   cmFinalRollerRearAxisX.commandConfiguration.phasing.phaseShiftChangeOnTheFly := FALSE;
   cmFinalRollerRearAxisX.commandConfiguration.offset.offset := 0.0;
   cmFinalRollerRearAxisX.commandConfiguration.offset.profileReference := 1;
   cmFinalRollerRearAxisX.commandConfiguration.offset.offsetDistance := 0.0;
   cmFinalRollerRearAxisX.commandConfiguration.offset.startPosition := 0.0;
   cmFinalRollerRearAxisX.commandConfiguration.offset.direction := 3;
   cmFinalRollerRearAxisX.commandConfiguration.offset.offsetAbsolute := TRUE;
   cmFinalRollerRearAxisX.commandConfiguration.offset.offsetChangeOnTheFly := FALSE;
   cmFinalRollerRearAxisX.commands.enableMasterControl := TRUE;
   cmFinalRollerRearAxisX.commands.enableAxis := FALSE;
   cmFinalRollerRearAxisX.commands.resetAxis := FALSE;
   cmFinalRollerRearAxisX.commands.openBrake := FALSE;
   cmFinalRollerRearAxisX.commands.jogForward := FALSE;
   cmFinalRollerRearAxisX.commands.jogBackward := FALSE;
   cmFinalRollerRearAxisX.commands.moveVelocity := FALSE;
   cmFinalRollerRearAxisX.commands.stop := FALSE;
   cmFinalRollerRearAxisX.commands.fastStop := FALSE;
   cmFinalRollerRearAxisX.commands.torqueLimiting := FALSE;
   cmFinalRollerRearAxisX.commands.homing := FALSE;
   cmFinalRollerRearAxisX.commands.posRelative := FALSE;
   cmFinalRollerRearAxisX.commands.posAbsolute := FALSE;
   cmFinalRollerRearAxisX.commands.posSuperimposed := FALSE;
   cmFinalRollerRearAxisX.commands.haltSuperimposed := FALSE;
   cmFinalRollerRearAxisX.commands.selectSetPosition := 0;
   cmFinalRollerRearAxisX.commands.uploadParameters := FALSE;
   cmFinalRollerRearAxisX.commands.refreshConfiguration := FALSE;
   cmFinalRollerRearAxisX.commands.editConfiguration := FALSE;
   cmFinalRollerRearAxisX.commands.saveConfiguration := FALSE;
   cmFinalRollerRearAxisX.commands.uploadCurrentTorque := FALSE;
   cmFinalRollerRearAxisX.commands.reset := FALSE;
   cmFinalRollerRearAxisX.monitoring.enable := TRUE;
   cmFinalRollerRearAxisX.monitoring.referenceDesignator := WSTRING#'FinalRollerRearAxisX';
   cmFinalRollerRearAxisX.monitoring.enabled := TRUE;
   cmFinalRollerRearAxisX.monitoring.enableManualCmds := FALSE;
   cmFinalRollerRearAxisX.monitoring.reset := FALSE;
   cmFinalRollerRearAxisX.monitoring.resetAxis := FALSE;
   cmFinalRollerRearAxisX.monitoring.enableAxis := TRUE;
   cmFinalRollerRearAxisX.monitoring.openBrake := FALSE;
   cmFinalRollerRearAxisX.monitoring.jogBackward := FALSE;
   cmFinalRollerRearAxisX.monitoring.jogForward := FALSE;
   cmFinalRollerRearAxisX.monitoring.moveVelocity := FALSE;
   cmFinalRollerRearAxisX.monitoring.stop := FALSE;
   cmFinalRollerRearAxisX.monitoring.fastStop := FALSE;
   cmFinalRollerRearAxisX.monitoring.torqueLimiting := FALSE;
   cmFinalRollerRearAxisX.monitoring.homing := FALSE;
   cmFinalRollerRearAxisX.monitoring.posRelative := FALSE;
   cmFinalRollerRearAxisX.monitoring.posAbsolute := FALSE;
   cmFinalRollerRearAxisX.monitoring.posSuperimposed := FALSE;
   cmFinalRollerRearAxisX.monitoring.haltSuperimposed := FALSE;
   cmFinalRollerRearAxisX.monitoring.brakeOpened := FALSE;
   cmFinalRollerRearAxisX.monitoring.axisEnabled := TRUE;
   cmFinalRollerRearAxisX.monitoring.resetActive := FALSE;
   cmFinalRollerRearAxisX.monitoring.inVelocity := FALSE;
   cmFinalRollerRearAxisX.monitoring.inLimitation := FALSE;
   cmFinalRollerRearAxisX.monitoring.inClamping := FALSE;
   cmFinalRollerRearAxisX.monitoring.startSync := FALSE;
   cmFinalRollerRearAxisX.monitoring.inSync := FALSE;
   cmFinalRollerRearAxisX.monitoring.inSimulation := FALSE;
   cmFinalRollerRearAxisX.monitoring.jogSelected := FALSE;
   cmFinalRollerRearAxisX.monitoring.moveVelocitySelected := FALSE;
   cmFinalRollerRearAxisX.monitoring.stopSelected := FALSE;
   cmFinalRollerRearAxisX.monitoring.fastStopSelected := FALSE;
   cmFinalRollerRearAxisX.monitoring.torqueLimitingSelected := FALSE;
   cmFinalRollerRearAxisX.monitoring.homingSelected := FALSE;
   cmFinalRollerRearAxisX.monitoring.posRelativeSelected := FALSE;
   cmFinalRollerRearAxisX.monitoring.posAbsoluteSelected := FALSE;
   cmFinalRollerRearAxisX.monitoring.posSuperimposedSelected := FALSE;
   cmFinalRollerRearAxisX.monitoring.haltSuperimposedSelected := FALSE;
   cmFinalRollerRearAxisX.monitoring.commandBusy := FALSE;
   cmFinalRollerRearAxisX.monitoring.commandDone := FALSE;
   cmFinalRollerRearAxisX.monitoring.commandAborted := FALSE;
   cmFinalRollerRearAxisX.monitoring.homingCommandBusy := FALSE;
   cmFinalRollerRearAxisX.monitoring.homingCommandDone := FALSE;
   cmFinalRollerRearAxisX.monitoring.homingCommandAborted := FALSE;
   cmFinalRollerRearAxisX.monitoring.superimposedBusy := FALSE;
   cmFinalRollerRearAxisX.monitoring.superimposedDone := FALSE;
   cmFinalRollerRearAxisX.monitoring.superimposedAborted := FALSE;
   cmFinalRollerRearAxisX.monitoring.selectSetPosition := 0;
   cmFinalRollerRearAxisX.monitoring.selectionController := FALSE;
   cmFinalRollerRearAxisX.monitoring.interlockGeneral := TRUE;
   cmFinalRollerRearAxisX.monitoring.interlockJogForward := TRUE;
   cmFinalRollerRearAxisX.monitoring.interlockJogBackward := TRUE;
   cmFinalRollerRearAxisX.monitoring.interlockWarningGeneral := FALSE;
   cmFinalRollerRearAxisX.monitoring.interlockWarningJogForward := FALSE;
   cmFinalRollerRearAxisX.monitoring.interlockWarningJogBackward := FALSE;
   cmFinalRollerRearAxisX.monitoring.valid := TRUE;
   cmFinalRollerRearAxisX.monitoring.busy := TRUE;
   cmFinalRollerRearAxisX.monitoring.error := FALSE;
   cmFinalRollerRearAxisX.monitoring.status := 16#7002;
   cmFinalRollerRearAxisX.monitoring.subfunctionStatus := 16#0000;
   cmFinalRollerRearAxisX.monitoring.actualPosition := 0.0;
   cmFinalRollerRearAxisX.monitoring.actualSpeed := 0.0;
   cmFinalRollerRearAxisX.monitoring.speedUnit := 1062;
   cmFinalRollerRearAxisX.monitoring.positionUnit := 1013;
   cmFinalRollerRearAxisX.monitoring.axisStatus1 := 16#0200_10E1;
   cmFinalRollerRearAxisX.monitoring.axisStatus2 := 16#0000_0000;
   cmFinalRollerRearAxisX.monitoring.axisType := 1;
   cmFinalRollerRearAxisX.monitoring.maxVelocity := 2500.0;
   cmFinalRollerRearAxisX.monitoring.actualCurrent := 0.0;
   cmFinalRollerRearAxisX.monitoring.actualTorque := 0.0;
   cmFinalRollerRearAxisX.monitoring.velocityOverrideEnabled := FALSE;
   cmFinalRollerRearAxisX.monitoring.sinaParaError := FALSE;
   cmFinalRollerRearAxisX.monitoring.sinaParaStatus := 16#0000_0000;
   cmFinalRollerRearAxisX.configuration.referenceDesignator := WSTRING#'FinalRollerRearAxisX';
   cmFinalRollerRearAxisX.configuration.disableAlarms := FALSE;
   cmFinalRollerRearAxisX.configuration.masterControlPopUp := TRUE;
   cmFinalRollerRearAxisX.configuration.setPositions[0].position := 0.0;
   cmFinalRollerRearAxisX.configuration.setPositions[1].position := 500.0;
   cmFinalRollerRearAxisX.configuration.setPositions[2..15].position := 0.0;
   cmFinalRollerRearAxisX.configuration.setPositions[0..1].velocity := 500.0;
   cmFinalRollerRearAxisX.configuration.setPositions[2..15].velocity := -1.0;
   cmFinalRollerRearAxisX.configuration.setPositions[0..1].acceleration := 5000.0;
   cmFinalRollerRearAxisX.configuration.setPositions[2..15].acceleration := -1.0;
   cmFinalRollerRearAxisX.configuration.setPositions[0..1].deceleration := 5000.0;
   cmFinalRollerRearAxisX.configuration.setPositions[2..15].deceleration := -1.0;
   cmFinalRollerRearAxisX.configuration.setPositions[0..15]."name" := '';
   cmMendrelAnodeFrontAxisY.commandConfiguration.generalSettings.stopOnError := TRUE;
   cmMendrelAnodeFrontAxisY.commandConfiguration.generalSettings.resetWithRestart := FALSE;
   cmMendrelAnodeFrontAxisY.commandConfiguration.generalSettings.abortWaitingSyncCmd := TRUE;
   cmMendrelAnodeFrontAxisY.commandConfiguration.power.startMode := 1;
   cmMendrelAnodeFrontAxisY.commandConfiguration.power.stopMode := 0;
   cmMendrelAnodeFrontAxisY.commandConfiguration.power.syncMotionSimulation := FALSE;
   cmMendrelAnodeFrontAxisY.commandConfiguration.power.syncMotionSimulationExtendedMode := -1;
   cmMendrelAnodeFrontAxisY.commandConfiguration.jog.velocity := 0.0;
   cmMendrelAnodeFrontAxisY.commandConfiguration.jog.acceleration := -1.0;
   cmMendrelAnodeFrontAxisY.commandConfiguration.jog.deceleration := -1.0;
   cmMendrelAnodeFrontAxisY.commandConfiguration.jog.jerk := -1.0;
   cmMendrelAnodeFrontAxisY.commandConfiguration.jog.positionControlled := TRUE;
   cmMendrelAnodeFrontAxisY.commandConfiguration.jog.increment := 0.0;
   cmMendrelAnodeFrontAxisY.commandConfiguration.jog.mode := 0;
   cmMendrelAnodeFrontAxisY.commandConfiguration.moveVelocity.velocity := 0.0;
   cmMendrelAnodeFrontAxisY.commandConfiguration.moveVelocity.acceleration := -1.0;
   cmMendrelAnodeFrontAxisY.commandConfiguration.moveVelocity.deceleration := -1.0;
   cmMendrelAnodeFrontAxisY.commandConfiguration.moveVelocity.jerk := -1.0;
   cmMendrelAnodeFrontAxisY.commandConfiguration.moveVelocity.direction := 0;
   cmMendrelAnodeFrontAxisY.commandConfiguration.moveVelocity.positionControlled := TRUE;
   cmMendrelAnodeFrontAxisY.commandConfiguration.moveVelocity.velocityChangeOnTheFly := FALSE;
   cmMendrelAnodeFrontAxisY.commandConfiguration.stop.deceleration := -1.0;
   cmMendrelAnodeFrontAxisY.commandConfiguration.stop.jerk := -1.0;
   cmMendrelAnodeFrontAxisY.commandConfiguration.stop.abortAcceleration := FALSE;
   cmMendrelAnodeFrontAxisY.commandConfiguration.fastStop.deceleration := -1.0;
   cmMendrelAnodeFrontAxisY.commandConfiguration.fastStop.jerk := -1.0;
   cmMendrelAnodeFrontAxisY.commandConfiguration.fastStop.abortAcceleration := FALSE;
   cmMendrelAnodeFrontAxisY.commandConfiguration.fastStop.replaceStopPossible := FALSE;
   cmMendrelAnodeFrontAxisY.commandConfiguration.torqueLimiting.limit := -1.0;
   cmMendrelAnodeFrontAxisY.commandConfiguration.torqueLimiting.mode := 0;
   cmMendrelAnodeFrontAxisY.commandConfiguration.homing.position := 0.0;
   cmMendrelAnodeFrontAxisY.commandConfiguration.homing.mode := 0;
   cmMendrelAnodeFrontAxisY.commandConfiguration.homing.sensor := 0;
   cmMendrelAnodeFrontAxisY.commandConfiguration.homing.extendedMode := -1;
   cmMendrelAnodeFrontAxisY.commandConfiguration.homing.extendedModeTorqueLimit := 0.0;
   cmMendrelAnodeFrontAxisY.commandConfiguration.homing.extendedModeTargetPosition := 0.0;
   cmMendrelAnodeFrontAxisY.commandConfiguration.posRelative.distance := 0.0;
   cmMendrelAnodeFrontAxisY.commandConfiguration.posRelative.velocity := -1.0;
   cmMendrelAnodeFrontAxisY.commandConfiguration.posRelative.acceleration := -1.0;
   cmMendrelAnodeFrontAxisY.commandConfiguration.posRelative.deceleration := -1.0;
   cmMendrelAnodeFrontAxisY.commandConfiguration.posRelative.jerk := -1.0;
   cmMendrelAnodeFrontAxisY.commandConfiguration.posRelative.direction := 0;
   cmMendrelAnodeFrontAxisY.commandConfiguration.posAbsolute.position := 0.0;
   cmMendrelAnodeFrontAxisY.commandConfiguration.posAbsolute.velocity := -1.0;
   cmMendrelAnodeFrontAxisY.commandConfiguration.posAbsolute.acceleration := -1.0;
   cmMendrelAnodeFrontAxisY.commandConfiguration.posAbsolute.deceleration := -1.0;
   cmMendrelAnodeFrontAxisY.commandConfiguration.posAbsolute.jerk := -1.0;
   cmMendrelAnodeFrontAxisY.commandConfiguration.posAbsolute.direction := 1;
   cmMendrelAnodeFrontAxisY.commandConfiguration.posAbsolute.positionChangeOnTheFly := FALSE;
   cmMendrelAnodeFrontAxisY.commandConfiguration.posAbsolute.velocityChangeOnTheFly := FALSE;
   cmMendrelAnodeFrontAxisY.commandConfiguration.posSuperimposed.distance := 0.0;
   cmMendrelAnodeFrontAxisY.commandConfiguration.posSuperimposed.velocityDiff := -1.0;
   cmMendrelAnodeFrontAxisY.commandConfiguration.posSuperimposed.acceleration := -1.0;
   cmMendrelAnodeFrontAxisY.commandConfiguration.posSuperimposed.deceleration := -1.0;
   cmMendrelAnodeFrontAxisY.commandConfiguration.posSuperimposed.jerk := -1.0;
   cmMendrelAnodeFrontAxisY.commandConfiguration.posSuperimposed.direction := 0;
   cmMendrelAnodeFrontAxisY.commandConfiguration.haltSuperimposed.deceleration := -1.0;
   cmMendrelAnodeFrontAxisY.commandConfiguration.haltSuperimposed.jerk := -1.0;
   cmMendrelAnodeFrontAxisY.commandConfiguration.haltSuperimposed.abortAcceleration := FALSE;
   cmMendrelAnodeFrontAxisY.commandConfiguration.gearInRelative.ratioNumerator := 1;
   cmMendrelAnodeFrontAxisY.commandConfiguration.gearInRelative.ratioDenominator := 1;
   cmMendrelAnodeFrontAxisY.commandConfiguration.gearInRelative.acceleration := -1.0;
   cmMendrelAnodeFrontAxisY.commandConfiguration.gearInRelative.deceleration := -1.0;
   cmMendrelAnodeFrontAxisY.commandConfiguration.gearInRelative.jerk := -1.0;
   cmMendrelAnodeFrontAxisY.commandConfiguration.gearInRelative.ratioChangeOnTheFly := FALSE;
   cmMendrelAnodeFrontAxisY.commandConfiguration.gearInAbsolute.ratioNumerator := 1;
   cmMendrelAnodeFrontAxisY.commandConfiguration.gearInAbsolute.ratioDenominator := 1;
   cmMendrelAnodeFrontAxisY.commandConfiguration.gearInAbsolute.masterSyncPosition := 0.0;
   cmMendrelAnodeFrontAxisY.commandConfiguration.gearInAbsolute.slaveSyncPosition := 0.0;
   cmMendrelAnodeFrontAxisY.commandConfiguration.gearInAbsolute.syncProfileReference := 1;
   cmMendrelAnodeFrontAxisY.commandConfiguration.gearInAbsolute.masterStartDistance := 0.0;
   cmMendrelAnodeFrontAxisY.commandConfiguration.gearInAbsolute.velocity := -1.0;
   cmMendrelAnodeFrontAxisY.commandConfiguration.gearInAbsolute.acceleration := -1.0;
   cmMendrelAnodeFrontAxisY.commandConfiguration.gearInAbsolute.deceleration := -1.0;
   cmMendrelAnodeFrontAxisY.commandConfiguration.gearInAbsolute.jerk := -1.0;
   cmMendrelAnodeFrontAxisY.commandConfiguration.gearInAbsolute.syncDirection := 1;
   cmMendrelAnodeFrontAxisY.commandConfiguration.gearInAbsolute.ratioChangeOnTheFly := FALSE;
   cmMendrelAnodeFrontAxisY.commandConfiguration.gearInVelocity.continuousUpdate := FALSE;
   cmMendrelAnodeFrontAxisY.commandConfiguration.gearInVelocity.ratioNumerator := 1;
   cmMendrelAnodeFrontAxisY.commandConfiguration.gearInVelocity.ratioDenominator := 1;
   cmMendrelAnodeFrontAxisY.commandConfiguration.gearInVelocity.acceleration := -1.0;
   cmMendrelAnodeFrontAxisY.commandConfiguration.gearInVelocity.deceleration := -1.0;
   cmMendrelAnodeFrontAxisY.commandConfiguration.gearInVelocity.jerk := -1.0;
   cmMendrelAnodeFrontAxisY.commandConfiguration.gearInVelocity.positionControlled := FALSE;
   cmMendrelAnodeFrontAxisY.commandConfiguration.camIn.masterOffset := 0.0;
   cmMendrelAnodeFrontAxisY.commandConfiguration.camIn.slaveOffset := 0.0;
   cmMendrelAnodeFrontAxisY.commandConfiguration.camIn.masterScaling := 1.0;
   cmMendrelAnodeFrontAxisY.commandConfiguration.camIn.slaveScaling := 1.0;
   cmMendrelAnodeFrontAxisY.commandConfiguration.camIn.masterSyncPosition := 0.0;
   cmMendrelAnodeFrontAxisY.commandConfiguration.camIn.syncProfileReference := 1;
   cmMendrelAnodeFrontAxisY.commandConfiguration.camIn.masterStartDistance := 0.0;
   cmMendrelAnodeFrontAxisY.commandConfiguration.camIn.velocity := -1.0;
   cmMendrelAnodeFrontAxisY.commandConfiguration.camIn.acceleration := -1.0;
   cmMendrelAnodeFrontAxisY.commandConfiguration.camIn.deceleration := -1.0;
   cmMendrelAnodeFrontAxisY.commandConfiguration.camIn.jerk := -1.0;
   cmMendrelAnodeFrontAxisY.commandConfiguration.camIn.applicationMode := 0;
   cmMendrelAnodeFrontAxisY.commandConfiguration.camIn.syncDirection := 1;
   cmMendrelAnodeFrontAxisY.commandConfiguration.gearOutCamOut.slavePosition := 0.0;
   cmMendrelAnodeFrontAxisY.commandConfiguration.gearOutCamOut.syncProfileReference := 1;
   cmMendrelAnodeFrontAxisY.commandConfiguration.gearOutCamOut.masterStopDistance := 0.0;
   cmMendrelAnodeFrontAxisY.commandConfiguration.gearOutCamOut.deceleration := -1.0;
   cmMendrelAnodeFrontAxisY.commandConfiguration.gearOutCamOut.jerk := -1.0;
   cmMendrelAnodeFrontAxisY.commandConfiguration.gearOutCamOut.syncOutDirection := 3;
   cmMendrelAnodeFrontAxisY.commandConfiguration.gearOutCamOut.gearOutCamOutMode := -1;
   cmMendrelAnodeFrontAxisY.commandConfiguration.phasing.phaseShift := 0.0;
   cmMendrelAnodeFrontAxisY.commandConfiguration.phasing.velocity := -1.0;
   cmMendrelAnodeFrontAxisY.commandConfiguration.phasing.acceleration := -1.0;
   cmMendrelAnodeFrontAxisY.commandConfiguration.phasing.deceleration := -1.0;
   cmMendrelAnodeFrontAxisY.commandConfiguration.phasing.jerk := -1.0;
   cmMendrelAnodeFrontAxisY.commandConfiguration.phasing.profileReference := 0;
   cmMendrelAnodeFrontAxisY.commandConfiguration.phasing.phasingDistance := 0.0;
   cmMendrelAnodeFrontAxisY.commandConfiguration.phasing.startPosition := 0.0;
   cmMendrelAnodeFrontAxisY.commandConfiguration.phasing.direction := 3;
   cmMendrelAnodeFrontAxisY.commandConfiguration.phasing.phaseAbsolute := TRUE;
   cmMendrelAnodeFrontAxisY.commandConfiguration.phasing.phaseShiftChangeOnTheFly := FALSE;
   cmMendrelAnodeFrontAxisY.commandConfiguration.offset.offset := 0.0;
   cmMendrelAnodeFrontAxisY.commandConfiguration.offset.profileReference := 1;
   cmMendrelAnodeFrontAxisY.commandConfiguration.offset.offsetDistance := 0.0;
   cmMendrelAnodeFrontAxisY.commandConfiguration.offset.startPosition := 0.0;
   cmMendrelAnodeFrontAxisY.commandConfiguration.offset.direction := 3;
   cmMendrelAnodeFrontAxisY.commandConfiguration.offset.offsetAbsolute := TRUE;
   cmMendrelAnodeFrontAxisY.commandConfiguration.offset.offsetChangeOnTheFly := FALSE;
   cmMendrelAnodeFrontAxisY.commands.enableMasterControl := TRUE;
   cmMendrelAnodeFrontAxisY.commands.enableAxis := FALSE;
   cmMendrelAnodeFrontAxisY.commands.resetAxis := FALSE;
   cmMendrelAnodeFrontAxisY.commands.openBrake := FALSE;
   cmMendrelAnodeFrontAxisY.commands.jogForward := FALSE;
   cmMendrelAnodeFrontAxisY.commands.jogBackward := FALSE;
   cmMendrelAnodeFrontAxisY.commands.moveVelocity := FALSE;
   cmMendrelAnodeFrontAxisY.commands.stop := FALSE;
   cmMendrelAnodeFrontAxisY.commands.fastStop := FALSE;
   cmMendrelAnodeFrontAxisY.commands.torqueLimiting := FALSE;
   cmMendrelAnodeFrontAxisY.commands.homing := FALSE;
   cmMendrelAnodeFrontAxisY.commands.posRelative := FALSE;
   cmMendrelAnodeFrontAxisY.commands.posAbsolute := FALSE;
   cmMendrelAnodeFrontAxisY.commands.posSuperimposed := FALSE;
   cmMendrelAnodeFrontAxisY.commands.haltSuperimposed := FALSE;
   cmMendrelAnodeFrontAxisY.commands.selectSetPosition := 1;
   cmMendrelAnodeFrontAxisY.commands.uploadParameters := FALSE;
   cmMendrelAnodeFrontAxisY.commands.refreshConfiguration := FALSE;
   cmMendrelAnodeFrontAxisY.commands.editConfiguration := FALSE;
   cmMendrelAnodeFrontAxisY.commands.saveConfiguration := FALSE;
   cmMendrelAnodeFrontAxisY.commands.uploadCurrentTorque := FALSE;
   cmMendrelAnodeFrontAxisY.commands.reset := FALSE;
   cmMendrelAnodeFrontAxisY.monitoring.enable := TRUE;
   cmMendrelAnodeFrontAxisY.monitoring.referenceDesignator := WSTRING#'MendrelAnodeFrontAxisY';
   cmMendrelAnodeFrontAxisY.monitoring.enabled := TRUE;
   cmMendrelAnodeFrontAxisY.monitoring.enableManualCmds := FALSE;
   cmMendrelAnodeFrontAxisY.monitoring.reset := FALSE;
   cmMendrelAnodeFrontAxisY.monitoring.resetAxis := FALSE;
   cmMendrelAnodeFrontAxisY.monitoring.enableAxis := TRUE;
   cmMendrelAnodeFrontAxisY.monitoring.openBrake := FALSE;
   cmMendrelAnodeFrontAxisY.monitoring.jogBackward := FALSE;
   cmMendrelAnodeFrontAxisY.monitoring.jogForward := FALSE;
   cmMendrelAnodeFrontAxisY.monitoring.moveVelocity := FALSE;
   cmMendrelAnodeFrontAxisY.monitoring.stop := FALSE;
   cmMendrelAnodeFrontAxisY.monitoring.fastStop := FALSE;
   cmMendrelAnodeFrontAxisY.monitoring.torqueLimiting := FALSE;
   cmMendrelAnodeFrontAxisY.monitoring.homing := FALSE;
   cmMendrelAnodeFrontAxisY.monitoring.posRelative := FALSE;
   cmMendrelAnodeFrontAxisY.monitoring.posAbsolute := FALSE;
   cmMendrelAnodeFrontAxisY.monitoring.posSuperimposed := FALSE;
   cmMendrelAnodeFrontAxisY.monitoring.haltSuperimposed := FALSE;
   cmMendrelAnodeFrontAxisY.monitoring.brakeOpened := FALSE;
   cmMendrelAnodeFrontAxisY.monitoring.axisEnabled := TRUE;
   cmMendrelAnodeFrontAxisY.monitoring.resetActive := FALSE;
   cmMendrelAnodeFrontAxisY.monitoring.inVelocity := FALSE;
   cmMendrelAnodeFrontAxisY.monitoring.inLimitation := FALSE;
   cmMendrelAnodeFrontAxisY.monitoring.inClamping := FALSE;
   cmMendrelAnodeFrontAxisY.monitoring.startSync := FALSE;
   cmMendrelAnodeFrontAxisY.monitoring.inSync := FALSE;
   cmMendrelAnodeFrontAxisY.monitoring.inSimulation := FALSE;
   cmMendrelAnodeFrontAxisY.monitoring.jogSelected := FALSE;
   cmMendrelAnodeFrontAxisY.monitoring.moveVelocitySelected := FALSE;
   cmMendrelAnodeFrontAxisY.monitoring.stopSelected := FALSE;
   cmMendrelAnodeFrontAxisY.monitoring.fastStopSelected := FALSE;
   cmMendrelAnodeFrontAxisY.monitoring.torqueLimitingSelected := FALSE;
   cmMendrelAnodeFrontAxisY.monitoring.homingSelected := FALSE;
   cmMendrelAnodeFrontAxisY.monitoring.posRelativeSelected := FALSE;
   cmMendrelAnodeFrontAxisY.monitoring.posAbsoluteSelected := FALSE;
   cmMendrelAnodeFrontAxisY.monitoring.posSuperimposedSelected := FALSE;
   cmMendrelAnodeFrontAxisY.monitoring.haltSuperimposedSelected := FALSE;
   cmMendrelAnodeFrontAxisY.monitoring.commandBusy := FALSE;
   cmMendrelAnodeFrontAxisY.monitoring.commandDone := FALSE;
   cmMendrelAnodeFrontAxisY.monitoring.commandAborted := FALSE;
   cmMendrelAnodeFrontAxisY.monitoring.homingCommandBusy := FALSE;
   cmMendrelAnodeFrontAxisY.monitoring.homingCommandDone := FALSE;
   cmMendrelAnodeFrontAxisY.monitoring.homingCommandAborted := FALSE;
   cmMendrelAnodeFrontAxisY.monitoring.superimposedBusy := FALSE;
   cmMendrelAnodeFrontAxisY.monitoring.superimposedDone := FALSE;
   cmMendrelAnodeFrontAxisY.monitoring.superimposedAborted := FALSE;
   cmMendrelAnodeFrontAxisY.monitoring.selectSetPosition := 1;
   cmMendrelAnodeFrontAxisY.monitoring.selectionController := FALSE;
   cmMendrelAnodeFrontAxisY.monitoring.interlockGeneral := TRUE;
   cmMendrelAnodeFrontAxisY.monitoring.interlockJogForward := TRUE;
   cmMendrelAnodeFrontAxisY.monitoring.interlockJogBackward := TRUE;
   cmMendrelAnodeFrontAxisY.monitoring.interlockWarningGeneral := FALSE;
   cmMendrelAnodeFrontAxisY.monitoring.interlockWarningJogForward := FALSE;
   cmMendrelAnodeFrontAxisY.monitoring.interlockWarningJogBackward := FALSE;
   cmMendrelAnodeFrontAxisY.monitoring.valid := TRUE;
   cmMendrelAnodeFrontAxisY.monitoring.busy := TRUE;
   cmMendrelAnodeFrontAxisY.monitoring.error := FALSE;
   cmMendrelAnodeFrontAxisY.monitoring.status := 16#7002;
   cmMendrelAnodeFrontAxisY.monitoring.subfunctionStatus := 16#0000;
   cmMendrelAnodeFrontAxisY.monitoring.actualPosition := 50.0;
   cmMendrelAnodeFrontAxisY.monitoring.actualSpeed := 0.0;
   cmMendrelAnodeFrontAxisY.monitoring.speedUnit := 1062;
   cmMendrelAnodeFrontAxisY.monitoring.positionUnit := 1013;
   cmMendrelAnodeFrontAxisY.monitoring.axisStatus1 := 16#0240_10A1;
   cmMendrelAnodeFrontAxisY.monitoring.axisStatus2 := 16#0000_0000;
   cmMendrelAnodeFrontAxisY.monitoring.axisType := 1;
   cmMendrelAnodeFrontAxisY.monitoring.maxVelocity := 2500.0;
   cmMendrelAnodeFrontAxisY.monitoring.actualCurrent := 0.0;
   cmMendrelAnodeFrontAxisY.monitoring.actualTorque := 0.0;
   cmMendrelAnodeFrontAxisY.monitoring.velocityOverrideEnabled := FALSE;
   cmMendrelAnodeFrontAxisY.monitoring.sinaParaError := FALSE;
   cmMendrelAnodeFrontAxisY.monitoring.sinaParaStatus := 16#0000_0000;
   cmMendrelAnodeFrontAxisY.configuration.referenceDesignator := WSTRING#'MendrelAnodeFrontAxisY';
   cmMendrelAnodeFrontAxisY.configuration.disableAlarms := FALSE;
   cmMendrelAnodeFrontAxisY.configuration.masterControlPopUp := TRUE;
   cmMendrelAnodeFrontAxisY.configuration.setPositions[0].position := 0.0;
   cmMendrelAnodeFrontAxisY.configuration.setPositions[1].position := 50.0;
   cmMendrelAnodeFrontAxisY.configuration.setPositions[2..15].position := 0.0;
   cmMendrelAnodeFrontAxisY.configuration.setPositions[0..1].velocity := 50.0;
   cmMendrelAnodeFrontAxisY.configuration.setPositions[2..15].velocity := -1.0;
   cmMendrelAnodeFrontAxisY.configuration.setPositions[0..1].acceleration := 500.0;
   cmMendrelAnodeFrontAxisY.configuration.setPositions[2..15].acceleration := -1.0;
   cmMendrelAnodeFrontAxisY.configuration.setPositions[0..1].deceleration := 500.0;
   cmMendrelAnodeFrontAxisY.configuration.setPositions[2..15].deceleration := -1.0;
   cmMendrelAnodeFrontAxisY.configuration.setPositions[0..15]."name" := '';
   cmMendrelAnodeFrontAxisZ.commandConfiguration.generalSettings.stopOnError := TRUE;
   cmMendrelAnodeFrontAxisZ.commandConfiguration.generalSettings.resetWithRestart := FALSE;
   cmMendrelAnodeFrontAxisZ.commandConfiguration.generalSettings.abortWaitingSyncCmd := TRUE;
   cmMendrelAnodeFrontAxisZ.commandConfiguration.power.startMode := 1;
   cmMendrelAnodeFrontAxisZ.commandConfiguration.power.stopMode := 0;
   cmMendrelAnodeFrontAxisZ.commandConfiguration.power.syncMotionSimulation := FALSE;
   cmMendrelAnodeFrontAxisZ.commandConfiguration.power.syncMotionSimulationExtendedMode := -1;
   cmMendrelAnodeFrontAxisZ.commandConfiguration.jog.velocity := 0.0;
   cmMendrelAnodeFrontAxisZ.commandConfiguration.jog.acceleration := -1.0;
   cmMendrelAnodeFrontAxisZ.commandConfiguration.jog.deceleration := -1.0;
   cmMendrelAnodeFrontAxisZ.commandConfiguration.jog.jerk := -1.0;
   cmMendrelAnodeFrontAxisZ.commandConfiguration.jog.positionControlled := TRUE;
   cmMendrelAnodeFrontAxisZ.commandConfiguration.jog.increment := 0.0;
   cmMendrelAnodeFrontAxisZ.commandConfiguration.jog.mode := 0;
   cmMendrelAnodeFrontAxisZ.commandConfiguration.moveVelocity.velocity := 0.0;
   cmMendrelAnodeFrontAxisZ.commandConfiguration.moveVelocity.acceleration := -1.0;
   cmMendrelAnodeFrontAxisZ.commandConfiguration.moveVelocity.deceleration := -1.0;
   cmMendrelAnodeFrontAxisZ.commandConfiguration.moveVelocity.jerk := -1.0;
   cmMendrelAnodeFrontAxisZ.commandConfiguration.moveVelocity.direction := 0;
   cmMendrelAnodeFrontAxisZ.commandConfiguration.moveVelocity.positionControlled := TRUE;
   cmMendrelAnodeFrontAxisZ.commandConfiguration.moveVelocity.velocityChangeOnTheFly := FALSE;
   cmMendrelAnodeFrontAxisZ.commandConfiguration.stop.deceleration := -1.0;
   cmMendrelAnodeFrontAxisZ.commandConfiguration.stop.jerk := -1.0;
   cmMendrelAnodeFrontAxisZ.commandConfiguration.stop.abortAcceleration := FALSE;
   cmMendrelAnodeFrontAxisZ.commandConfiguration.fastStop.deceleration := -1.0;
   cmMendrelAnodeFrontAxisZ.commandConfiguration.fastStop.jerk := -1.0;
   cmMendrelAnodeFrontAxisZ.commandConfiguration.fastStop.abortAcceleration := FALSE;
   cmMendrelAnodeFrontAxisZ.commandConfiguration.fastStop.replaceStopPossible := FALSE;
   cmMendrelAnodeFrontAxisZ.commandConfiguration.torqueLimiting.limit := -1.0;
   cmMendrelAnodeFrontAxisZ.commandConfiguration.torqueLimiting.mode := 0;
   cmMendrelAnodeFrontAxisZ.commandConfiguration.homing.position := 0.0;
   cmMendrelAnodeFrontAxisZ.commandConfiguration.homing.mode := 0;
   cmMendrelAnodeFrontAxisZ.commandConfiguration.homing.sensor := 0;
   cmMendrelAnodeFrontAxisZ.commandConfiguration.homing.extendedMode := -1;
   cmMendrelAnodeFrontAxisZ.commandConfiguration.homing.extendedModeTorqueLimit := 0.0;
   cmMendrelAnodeFrontAxisZ.commandConfiguration.homing.extendedModeTargetPosition := 0.0;
   cmMendrelAnodeFrontAxisZ.commandConfiguration.posRelative.distance := 0.0;
   cmMendrelAnodeFrontAxisZ.commandConfiguration.posRelative.velocity := -1.0;
   cmMendrelAnodeFrontAxisZ.commandConfiguration.posRelative.acceleration := -1.0;
   cmMendrelAnodeFrontAxisZ.commandConfiguration.posRelative.deceleration := -1.0;
   cmMendrelAnodeFrontAxisZ.commandConfiguration.posRelative.jerk := -1.0;
   cmMendrelAnodeFrontAxisZ.commandConfiguration.posRelative.direction := 0;
   cmMendrelAnodeFrontAxisZ.commandConfiguration.posAbsolute.position := 0.0;
   cmMendrelAnodeFrontAxisZ.commandConfiguration.posAbsolute.velocity := -1.0;
   cmMendrelAnodeFrontAxisZ.commandConfiguration.posAbsolute.acceleration := -1.0;
   cmMendrelAnodeFrontAxisZ.commandConfiguration.posAbsolute.deceleration := -1.0;
   cmMendrelAnodeFrontAxisZ.commandConfiguration.posAbsolute.jerk := -1.0;
   cmMendrelAnodeFrontAxisZ.commandConfiguration.posAbsolute.direction := 1;
   cmMendrelAnodeFrontAxisZ.commandConfiguration.posAbsolute.positionChangeOnTheFly := FALSE;
   cmMendrelAnodeFrontAxisZ.commandConfiguration.posAbsolute.velocityChangeOnTheFly := FALSE;
   cmMendrelAnodeFrontAxisZ.commandConfiguration.posSuperimposed.distance := 0.0;
   cmMendrelAnodeFrontAxisZ.commandConfiguration.posSuperimposed.velocityDiff := -1.0;
   cmMendrelAnodeFrontAxisZ.commandConfiguration.posSuperimposed.acceleration := -1.0;
   cmMendrelAnodeFrontAxisZ.commandConfiguration.posSuperimposed.deceleration := -1.0;
   cmMendrelAnodeFrontAxisZ.commandConfiguration.posSuperimposed.jerk := -1.0;
   cmMendrelAnodeFrontAxisZ.commandConfiguration.posSuperimposed.direction := 0;
   cmMendrelAnodeFrontAxisZ.commandConfiguration.haltSuperimposed.deceleration := -1.0;
   cmMendrelAnodeFrontAxisZ.commandConfiguration.haltSuperimposed.jerk := -1.0;
   cmMendrelAnodeFrontAxisZ.commandConfiguration.haltSuperimposed.abortAcceleration := FALSE;
   cmMendrelAnodeFrontAxisZ.commandConfiguration.gearInRelative.ratioNumerator := 1;
   cmMendrelAnodeFrontAxisZ.commandConfiguration.gearInRelative.ratioDenominator := 1;
   cmMendrelAnodeFrontAxisZ.commandConfiguration.gearInRelative.acceleration := -1.0;
   cmMendrelAnodeFrontAxisZ.commandConfiguration.gearInRelative.deceleration := -1.0;
   cmMendrelAnodeFrontAxisZ.commandConfiguration.gearInRelative.jerk := -1.0;
   cmMendrelAnodeFrontAxisZ.commandConfiguration.gearInRelative.ratioChangeOnTheFly := FALSE;
   cmMendrelAnodeFrontAxisZ.commandConfiguration.gearInAbsolute.ratioNumerator := 1;
   cmMendrelAnodeFrontAxisZ.commandConfiguration.gearInAbsolute.ratioDenominator := 1;
   cmMendrelAnodeFrontAxisZ.commandConfiguration.gearInAbsolute.masterSyncPosition := 0.0;
   cmMendrelAnodeFrontAxisZ.commandConfiguration.gearInAbsolute.slaveSyncPosition := 0.0;
   cmMendrelAnodeFrontAxisZ.commandConfiguration.gearInAbsolute.syncProfileReference := 1;
   cmMendrelAnodeFrontAxisZ.commandConfiguration.gearInAbsolute.masterStartDistance := 0.0;
   cmMendrelAnodeFrontAxisZ.commandConfiguration.gearInAbsolute.velocity := -1.0;
   cmMendrelAnodeFrontAxisZ.commandConfiguration.gearInAbsolute.acceleration := -1.0;
   cmMendrelAnodeFrontAxisZ.commandConfiguration.gearInAbsolute.deceleration := -1.0;
   cmMendrelAnodeFrontAxisZ.commandConfiguration.gearInAbsolute.jerk := -1.0;
   cmMendrelAnodeFrontAxisZ.commandConfiguration.gearInAbsolute.syncDirection := 1;
   cmMendrelAnodeFrontAxisZ.commandConfiguration.gearInAbsolute.ratioChangeOnTheFly := FALSE;
   cmMendrelAnodeFrontAxisZ.commandConfiguration.gearInVelocity.continuousUpdate := FALSE;
   cmMendrelAnodeFrontAxisZ.commandConfiguration.gearInVelocity.ratioNumerator := 1;
   cmMendrelAnodeFrontAxisZ.commandConfiguration.gearInVelocity.ratioDenominator := 1;
   cmMendrelAnodeFrontAxisZ.commandConfiguration.gearInVelocity.acceleration := -1.0;
   cmMendrelAnodeFrontAxisZ.commandConfiguration.gearInVelocity.deceleration := -1.0;
   cmMendrelAnodeFrontAxisZ.commandConfiguration.gearInVelocity.jerk := -1.0;
   cmMendrelAnodeFrontAxisZ.commandConfiguration.gearInVelocity.positionControlled := FALSE;
   cmMendrelAnodeFrontAxisZ.commandConfiguration.camIn.masterOffset := 0.0;
   cmMendrelAnodeFrontAxisZ.commandConfiguration.camIn.slaveOffset := 0.0;
   cmMendrelAnodeFrontAxisZ.commandConfiguration.camIn.masterScaling := 1.0;
   cmMendrelAnodeFrontAxisZ.commandConfiguration.camIn.slaveScaling := 1.0;
   cmMendrelAnodeFrontAxisZ.commandConfiguration.camIn.masterSyncPosition := 0.0;
   cmMendrelAnodeFrontAxisZ.commandConfiguration.camIn.syncProfileReference := 1;
   cmMendrelAnodeFrontAxisZ.commandConfiguration.camIn.masterStartDistance := 0.0;
   cmMendrelAnodeFrontAxisZ.commandConfiguration.camIn.velocity := -1.0;
   cmMendrelAnodeFrontAxisZ.commandConfiguration.camIn.acceleration := -1.0;
   cmMendrelAnodeFrontAxisZ.commandConfiguration.camIn.deceleration := -1.0;
   cmMendrelAnodeFrontAxisZ.commandConfiguration.camIn.jerk := -1.0;
   cmMendrelAnodeFrontAxisZ.commandConfiguration.camIn.applicationMode := 0;
   cmMendrelAnodeFrontAxisZ.commandConfiguration.camIn.syncDirection := 1;
   cmMendrelAnodeFrontAxisZ.commandConfiguration.gearOutCamOut.slavePosition := 0.0;
   cmMendrelAnodeFrontAxisZ.commandConfiguration.gearOutCamOut.syncProfileReference := 1;
   cmMendrelAnodeFrontAxisZ.commandConfiguration.gearOutCamOut.masterStopDistance := 0.0;
   cmMendrelAnodeFrontAxisZ.commandConfiguration.gearOutCamOut.deceleration := -1.0;
   cmMendrelAnodeFrontAxisZ.commandConfiguration.gearOutCamOut.jerk := -1.0;
   cmMendrelAnodeFrontAxisZ.commandConfiguration.gearOutCamOut.syncOutDirection := 3;
   cmMendrelAnodeFrontAxisZ.commandConfiguration.gearOutCamOut.gearOutCamOutMode := -1;
   cmMendrelAnodeFrontAxisZ.commandConfiguration.phasing.phaseShift := 0.0;
   cmMendrelAnodeFrontAxisZ.commandConfiguration.phasing.velocity := -1.0;
   cmMendrelAnodeFrontAxisZ.commandConfiguration.phasing.acceleration := -1.0;
   cmMendrelAnodeFrontAxisZ.commandConfiguration.phasing.deceleration := -1.0;
   cmMendrelAnodeFrontAxisZ.commandConfiguration.phasing.jerk := -1.0;
   cmMendrelAnodeFrontAxisZ.commandConfiguration.phasing.profileReference := 0;
   cmMendrelAnodeFrontAxisZ.commandConfiguration.phasing.phasingDistance := 0.0;
   cmMendrelAnodeFrontAxisZ.commandConfiguration.phasing.startPosition := 0.0;
   cmMendrelAnodeFrontAxisZ.commandConfiguration.phasing.direction := 3;
   cmMendrelAnodeFrontAxisZ.commandConfiguration.phasing.phaseAbsolute := TRUE;
   cmMendrelAnodeFrontAxisZ.commandConfiguration.phasing.phaseShiftChangeOnTheFly := FALSE;
   cmMendrelAnodeFrontAxisZ.commandConfiguration.offset.offset := 0.0;
   cmMendrelAnodeFrontAxisZ.commandConfiguration.offset.profileReference := 1;
   cmMendrelAnodeFrontAxisZ.commandConfiguration.offset.offsetDistance := 0.0;
   cmMendrelAnodeFrontAxisZ.commandConfiguration.offset.startPosition := 0.0;
   cmMendrelAnodeFrontAxisZ.commandConfiguration.offset.direction := 3;
   cmMendrelAnodeFrontAxisZ.commandConfiguration.offset.offsetAbsolute := TRUE;
   cmMendrelAnodeFrontAxisZ.commandConfiguration.offset.offsetChangeOnTheFly := FALSE;
   cmMendrelAnodeFrontAxisZ.commands.enableMasterControl := TRUE;
   cmMendrelAnodeFrontAxisZ.commands.enableAxis := FALSE;
   cmMendrelAnodeFrontAxisZ.commands.resetAxis := FALSE;
   cmMendrelAnodeFrontAxisZ.commands.openBrake := FALSE;
   cmMendrelAnodeFrontAxisZ.commands.jogForward := FALSE;
   cmMendrelAnodeFrontAxisZ.commands.jogBackward := FALSE;
   cmMendrelAnodeFrontAxisZ.commands.moveVelocity := FALSE;
   cmMendrelAnodeFrontAxisZ.commands.stop := FALSE;
   cmMendrelAnodeFrontAxisZ.commands.fastStop := FALSE;
   cmMendrelAnodeFrontAxisZ.commands.torqueLimiting := FALSE;
   cmMendrelAnodeFrontAxisZ.commands.homing := FALSE;
   cmMendrelAnodeFrontAxisZ.commands.posRelative := FALSE;
   cmMendrelAnodeFrontAxisZ.commands.posAbsolute := FALSE;
   cmMendrelAnodeFrontAxisZ.commands.posSuperimposed := FALSE;
   cmMendrelAnodeFrontAxisZ.commands.haltSuperimposed := FALSE;
   cmMendrelAnodeFrontAxisZ.commands.selectSetPosition := 1;
   cmMendrelAnodeFrontAxisZ.commands.uploadParameters := FALSE;
   cmMendrelAnodeFrontAxisZ.commands.refreshConfiguration := FALSE;
   cmMendrelAnodeFrontAxisZ.commands.editConfiguration := FALSE;
   cmMendrelAnodeFrontAxisZ.commands.saveConfiguration := FALSE;
   cmMendrelAnodeFrontAxisZ.commands.uploadCurrentTorque := FALSE;
   cmMendrelAnodeFrontAxisZ.commands.reset := FALSE;
   cmMendrelAnodeFrontAxisZ.monitoring.enable := TRUE;
   cmMendrelAnodeFrontAxisZ.monitoring.referenceDesignator := WSTRING#'MendrelAnodeFrontAxisZ';
   cmMendrelAnodeFrontAxisZ.monitoring.enabled := TRUE;
   cmMendrelAnodeFrontAxisZ.monitoring.enableManualCmds := FALSE;
   cmMendrelAnodeFrontAxisZ.monitoring.reset := FALSE;
   cmMendrelAnodeFrontAxisZ.monitoring.resetAxis := FALSE;
   cmMendrelAnodeFrontAxisZ.monitoring.enableAxis := TRUE;
   cmMendrelAnodeFrontAxisZ.monitoring.openBrake := FALSE;
   cmMendrelAnodeFrontAxisZ.monitoring.jogBackward := FALSE;
   cmMendrelAnodeFrontAxisZ.monitoring.jogForward := FALSE;
   cmMendrelAnodeFrontAxisZ.monitoring.moveVelocity := FALSE;
   cmMendrelAnodeFrontAxisZ.monitoring.stop := FALSE;
   cmMendrelAnodeFrontAxisZ.monitoring.fastStop := FALSE;
   cmMendrelAnodeFrontAxisZ.monitoring.torqueLimiting := FALSE;
   cmMendrelAnodeFrontAxisZ.monitoring.homing := FALSE;
   cmMendrelAnodeFrontAxisZ.monitoring.posRelative := FALSE;
   cmMendrelAnodeFrontAxisZ.monitoring.posAbsolute := FALSE;
   cmMendrelAnodeFrontAxisZ.monitoring.posSuperimposed := FALSE;
   cmMendrelAnodeFrontAxisZ.monitoring.haltSuperimposed := FALSE;
   cmMendrelAnodeFrontAxisZ.monitoring.brakeOpened := FALSE;
   cmMendrelAnodeFrontAxisZ.monitoring.axisEnabled := TRUE;
   cmMendrelAnodeFrontAxisZ.monitoring.resetActive := FALSE;
   cmMendrelAnodeFrontAxisZ.monitoring.inVelocity := FALSE;
   cmMendrelAnodeFrontAxisZ.monitoring.inLimitation := FALSE;
   cmMendrelAnodeFrontAxisZ.monitoring.inClamping := FALSE;
   cmMendrelAnodeFrontAxisZ.monitoring.startSync := FALSE;
   cmMendrelAnodeFrontAxisZ.monitoring.inSync := FALSE;
   cmMendrelAnodeFrontAxisZ.monitoring.inSimulation := FALSE;
   cmMendrelAnodeFrontAxisZ.monitoring.jogSelected := FALSE;
   cmMendrelAnodeFrontAxisZ.monitoring.moveVelocitySelected := FALSE;
   cmMendrelAnodeFrontAxisZ.monitoring.stopSelected := FALSE;
   cmMendrelAnodeFrontAxisZ.monitoring.fastStopSelected := FALSE;
   cmMendrelAnodeFrontAxisZ.monitoring.torqueLimitingSelected := FALSE;
   cmMendrelAnodeFrontAxisZ.monitoring.homingSelected := FALSE;
   cmMendrelAnodeFrontAxisZ.monitoring.posRelativeSelected := FALSE;
   cmMendrelAnodeFrontAxisZ.monitoring.posAbsoluteSelected := FALSE;
   cmMendrelAnodeFrontAxisZ.monitoring.posSuperimposedSelected := FALSE;
   cmMendrelAnodeFrontAxisZ.monitoring.haltSuperimposedSelected := FALSE;
   cmMendrelAnodeFrontAxisZ.monitoring.commandBusy := FALSE;
   cmMendrelAnodeFrontAxisZ.monitoring.commandDone := FALSE;
   cmMendrelAnodeFrontAxisZ.monitoring.commandAborted := FALSE;
   cmMendrelAnodeFrontAxisZ.monitoring.homingCommandBusy := FALSE;
   cmMendrelAnodeFrontAxisZ.monitoring.homingCommandDone := FALSE;
   cmMendrelAnodeFrontAxisZ.monitoring.homingCommandAborted := FALSE;
   cmMendrelAnodeFrontAxisZ.monitoring.superimposedBusy := FALSE;
   cmMendrelAnodeFrontAxisZ.monitoring.superimposedDone := FALSE;
   cmMendrelAnodeFrontAxisZ.monitoring.superimposedAborted := FALSE;
   cmMendrelAnodeFrontAxisZ.monitoring.selectSetPosition := 1;
   cmMendrelAnodeFrontAxisZ.monitoring.selectionController := FALSE;
   cmMendrelAnodeFrontAxisZ.monitoring.interlockGeneral := TRUE;
   cmMendrelAnodeFrontAxisZ.monitoring.interlockJogForward := TRUE;
   cmMendrelAnodeFrontAxisZ.monitoring.interlockJogBackward := TRUE;
   cmMendrelAnodeFrontAxisZ.monitoring.interlockWarningGeneral := FALSE;
   cmMendrelAnodeFrontAxisZ.monitoring.interlockWarningJogForward := FALSE;
   cmMendrelAnodeFrontAxisZ.monitoring.interlockWarningJogBackward := FALSE;
   cmMendrelAnodeFrontAxisZ.monitoring.valid := TRUE;
   cmMendrelAnodeFrontAxisZ.monitoring.busy := TRUE;
   cmMendrelAnodeFrontAxisZ.monitoring.error := FALSE;
   cmMendrelAnodeFrontAxisZ.monitoring.status := 16#7002;
   cmMendrelAnodeFrontAxisZ.monitoring.subfunctionStatus := 16#0000;
   cmMendrelAnodeFrontAxisZ.monitoring.actualPosition := 50.0;
   cmMendrelAnodeFrontAxisZ.monitoring.actualSpeed := 0.0;
   cmMendrelAnodeFrontAxisZ.monitoring.speedUnit := 1062;
   cmMendrelAnodeFrontAxisZ.monitoring.positionUnit := 1013;
   cmMendrelAnodeFrontAxisZ.monitoring.axisStatus1 := 16#0240_10A1;
   cmMendrelAnodeFrontAxisZ.monitoring.axisStatus2 := 16#0000_0000;
   cmMendrelAnodeFrontAxisZ.monitoring.axisType := 1;
   cmMendrelAnodeFrontAxisZ.monitoring.maxVelocity := 2500.0;
   cmMendrelAnodeFrontAxisZ.monitoring.actualCurrent := 0.0;
   cmMendrelAnodeFrontAxisZ.monitoring.actualTorque := 0.0;
   cmMendrelAnodeFrontAxisZ.monitoring.velocityOverrideEnabled := FALSE;
   cmMendrelAnodeFrontAxisZ.monitoring.sinaParaError := FALSE;
   cmMendrelAnodeFrontAxisZ.monitoring.sinaParaStatus := 16#0000_0000;
   cmMendrelAnodeFrontAxisZ.configuration.referenceDesignator := WSTRING#'MendrelAnodeFrontAxisZ';
   cmMendrelAnodeFrontAxisZ.configuration.disableAlarms := FALSE;
   cmMendrelAnodeFrontAxisZ.configuration.masterControlPopUp := TRUE;
   cmMendrelAnodeFrontAxisZ.configuration.setPositions[0].position := 0.0;
   cmMendrelAnodeFrontAxisZ.configuration.setPositions[1].position := 50.0;
   cmMendrelAnodeFrontAxisZ.configuration.setPositions[2..15].position := 0.0;
   cmMendrelAnodeFrontAxisZ.configuration.setPositions[0..1].velocity := 50.0;
   cmMendrelAnodeFrontAxisZ.configuration.setPositions[2..15].velocity := -1.0;
   cmMendrelAnodeFrontAxisZ.configuration.setPositions[0..1].acceleration := 500.0;
   cmMendrelAnodeFrontAxisZ.configuration.setPositions[2..15].acceleration := -1.0;
   cmMendrelAnodeFrontAxisZ.configuration.setPositions[0..1].deceleration := 500.0;
   cmMendrelAnodeFrontAxisZ.configuration.setPositions[2..15].deceleration := -1.0;
   cmMendrelAnodeFrontAxisZ.configuration.setPositions[0..15]."name" := '';
   cmMendrelAnodeRearAxisY.commandConfiguration.generalSettings.stopOnError := TRUE;
   cmMendrelAnodeRearAxisY.commandConfiguration.generalSettings.resetWithRestart := FALSE;
   cmMendrelAnodeRearAxisY.commandConfiguration.generalSettings.abortWaitingSyncCmd := TRUE;
   cmMendrelAnodeRearAxisY.commandConfiguration.power.startMode := 1;
   cmMendrelAnodeRearAxisY.commandConfiguration.power.stopMode := 0;
   cmMendrelAnodeRearAxisY.commandConfiguration.power.syncMotionSimulation := FALSE;
   cmMendrelAnodeRearAxisY.commandConfiguration.power.syncMotionSimulationExtendedMode := -1;
   cmMendrelAnodeRearAxisY.commandConfiguration.jog.velocity := 0.0;
   cmMendrelAnodeRearAxisY.commandConfiguration.jog.acceleration := -1.0;
   cmMendrelAnodeRearAxisY.commandConfiguration.jog.deceleration := -1.0;
   cmMendrelAnodeRearAxisY.commandConfiguration.jog.jerk := -1.0;
   cmMendrelAnodeRearAxisY.commandConfiguration.jog.positionControlled := TRUE;
   cmMendrelAnodeRearAxisY.commandConfiguration.jog.increment := 0.0;
   cmMendrelAnodeRearAxisY.commandConfiguration.jog.mode := 0;
   cmMendrelAnodeRearAxisY.commandConfiguration.moveVelocity.velocity := 0.0;
   cmMendrelAnodeRearAxisY.commandConfiguration.moveVelocity.acceleration := -1.0;
   cmMendrelAnodeRearAxisY.commandConfiguration.moveVelocity.deceleration := -1.0;
   cmMendrelAnodeRearAxisY.commandConfiguration.moveVelocity.jerk := -1.0;
   cmMendrelAnodeRearAxisY.commandConfiguration.moveVelocity.direction := 0;
   cmMendrelAnodeRearAxisY.commandConfiguration.moveVelocity.positionControlled := TRUE;
   cmMendrelAnodeRearAxisY.commandConfiguration.moveVelocity.velocityChangeOnTheFly := FALSE;
   cmMendrelAnodeRearAxisY.commandConfiguration.stop.deceleration := -1.0;
   cmMendrelAnodeRearAxisY.commandConfiguration.stop.jerk := -1.0;
   cmMendrelAnodeRearAxisY.commandConfiguration.stop.abortAcceleration := FALSE;
   cmMendrelAnodeRearAxisY.commandConfiguration.fastStop.deceleration := -1.0;
   cmMendrelAnodeRearAxisY.commandConfiguration.fastStop.jerk := -1.0;
   cmMendrelAnodeRearAxisY.commandConfiguration.fastStop.abortAcceleration := FALSE;
   cmMendrelAnodeRearAxisY.commandConfiguration.fastStop.replaceStopPossible := FALSE;
   cmMendrelAnodeRearAxisY.commandConfiguration.torqueLimiting.limit := -1.0;
   cmMendrelAnodeRearAxisY.commandConfiguration.torqueLimiting.mode := 0;
   cmMendrelAnodeRearAxisY.commandConfiguration.homing.position := 0.0;
   cmMendrelAnodeRearAxisY.commandConfiguration.homing.mode := 0;
   cmMendrelAnodeRearAxisY.commandConfiguration.homing.sensor := 0;
   cmMendrelAnodeRearAxisY.commandConfiguration.homing.extendedMode := -1;
   cmMendrelAnodeRearAxisY.commandConfiguration.homing.extendedModeTorqueLimit := 0.0;
   cmMendrelAnodeRearAxisY.commandConfiguration.homing.extendedModeTargetPosition := 0.0;
   cmMendrelAnodeRearAxisY.commandConfiguration.posRelative.distance := 0.0;
   cmMendrelAnodeRearAxisY.commandConfiguration.posRelative.velocity := -1.0;
   cmMendrelAnodeRearAxisY.commandConfiguration.posRelative.acceleration := -1.0;
   cmMendrelAnodeRearAxisY.commandConfiguration.posRelative.deceleration := -1.0;
   cmMendrelAnodeRearAxisY.commandConfiguration.posRelative.jerk := -1.0;
   cmMendrelAnodeRearAxisY.commandConfiguration.posRelative.direction := 0;
   cmMendrelAnodeRearAxisY.commandConfiguration.posAbsolute.position := 0.0;
   cmMendrelAnodeRearAxisY.commandConfiguration.posAbsolute.velocity := -1.0;
   cmMendrelAnodeRearAxisY.commandConfiguration.posAbsolute.acceleration := -1.0;
   cmMendrelAnodeRearAxisY.commandConfiguration.posAbsolute.deceleration := -1.0;
   cmMendrelAnodeRearAxisY.commandConfiguration.posAbsolute.jerk := -1.0;
   cmMendrelAnodeRearAxisY.commandConfiguration.posAbsolute.direction := 1;
   cmMendrelAnodeRearAxisY.commandConfiguration.posAbsolute.positionChangeOnTheFly := FALSE;
   cmMendrelAnodeRearAxisY.commandConfiguration.posAbsolute.velocityChangeOnTheFly := FALSE;
   cmMendrelAnodeRearAxisY.commandConfiguration.posSuperimposed.distance := 0.0;
   cmMendrelAnodeRearAxisY.commandConfiguration.posSuperimposed.velocityDiff := -1.0;
   cmMendrelAnodeRearAxisY.commandConfiguration.posSuperimposed.acceleration := -1.0;
   cmMendrelAnodeRearAxisY.commandConfiguration.posSuperimposed.deceleration := -1.0;
   cmMendrelAnodeRearAxisY.commandConfiguration.posSuperimposed.jerk := -1.0;
   cmMendrelAnodeRearAxisY.commandConfiguration.posSuperimposed.direction := 0;
   cmMendrelAnodeRearAxisY.commandConfiguration.haltSuperimposed.deceleration := -1.0;
   cmMendrelAnodeRearAxisY.commandConfiguration.haltSuperimposed.jerk := -1.0;
   cmMendrelAnodeRearAxisY.commandConfiguration.haltSuperimposed.abortAcceleration := FALSE;
   cmMendrelAnodeRearAxisY.commandConfiguration.gearInRelative.ratioNumerator := 1;
   cmMendrelAnodeRearAxisY.commandConfiguration.gearInRelative.ratioDenominator := 1;
   cmMendrelAnodeRearAxisY.commandConfiguration.gearInRelative.acceleration := -1.0;
   cmMendrelAnodeRearAxisY.commandConfiguration.gearInRelative.deceleration := -1.0;
   cmMendrelAnodeRearAxisY.commandConfiguration.gearInRelative.jerk := -1.0;
   cmMendrelAnodeRearAxisY.commandConfiguration.gearInRelative.ratioChangeOnTheFly := FALSE;
   cmMendrelAnodeRearAxisY.commandConfiguration.gearInAbsolute.ratioNumerator := 1;
   cmMendrelAnodeRearAxisY.commandConfiguration.gearInAbsolute.ratioDenominator := 1;
   cmMendrelAnodeRearAxisY.commandConfiguration.gearInAbsolute.masterSyncPosition := 0.0;
   cmMendrelAnodeRearAxisY.commandConfiguration.gearInAbsolute.slaveSyncPosition := 0.0;
   cmMendrelAnodeRearAxisY.commandConfiguration.gearInAbsolute.syncProfileReference := 1;
   cmMendrelAnodeRearAxisY.commandConfiguration.gearInAbsolute.masterStartDistance := 0.0;
   cmMendrelAnodeRearAxisY.commandConfiguration.gearInAbsolute.velocity := -1.0;
   cmMendrelAnodeRearAxisY.commandConfiguration.gearInAbsolute.acceleration := -1.0;
   cmMendrelAnodeRearAxisY.commandConfiguration.gearInAbsolute.deceleration := -1.0;
   cmMendrelAnodeRearAxisY.commandConfiguration.gearInAbsolute.jerk := -1.0;
   cmMendrelAnodeRearAxisY.commandConfiguration.gearInAbsolute.syncDirection := 1;
   cmMendrelAnodeRearAxisY.commandConfiguration.gearInAbsolute.ratioChangeOnTheFly := FALSE;
   cmMendrelAnodeRearAxisY.commandConfiguration.gearInVelocity.continuousUpdate := FALSE;
   cmMendrelAnodeRearAxisY.commandConfiguration.gearInVelocity.ratioNumerator := 1;
   cmMendrelAnodeRearAxisY.commandConfiguration.gearInVelocity.ratioDenominator := 1;
   cmMendrelAnodeRearAxisY.commandConfiguration.gearInVelocity.acceleration := -1.0;
   cmMendrelAnodeRearAxisY.commandConfiguration.gearInVelocity.deceleration := -1.0;
   cmMendrelAnodeRearAxisY.commandConfiguration.gearInVelocity.jerk := -1.0;
   cmMendrelAnodeRearAxisY.commandConfiguration.gearInVelocity.positionControlled := FALSE;
   cmMendrelAnodeRearAxisY.commandConfiguration.camIn.masterOffset := 0.0;
   cmMendrelAnodeRearAxisY.commandConfiguration.camIn.slaveOffset := 0.0;
   cmMendrelAnodeRearAxisY.commandConfiguration.camIn.masterScaling := 1.0;
   cmMendrelAnodeRearAxisY.commandConfiguration.camIn.slaveScaling := 1.0;
   cmMendrelAnodeRearAxisY.commandConfiguration.camIn.masterSyncPosition := 0.0;
   cmMendrelAnodeRearAxisY.commandConfiguration.camIn.syncProfileReference := 1;
   cmMendrelAnodeRearAxisY.commandConfiguration.camIn.masterStartDistance := 0.0;
   cmMendrelAnodeRearAxisY.commandConfiguration.camIn.velocity := -1.0;
   cmMendrelAnodeRearAxisY.commandConfiguration.camIn.acceleration := -1.0;
   cmMendrelAnodeRearAxisY.commandConfiguration.camIn.deceleration := -1.0;
   cmMendrelAnodeRearAxisY.commandConfiguration.camIn.jerk := -1.0;
   cmMendrelAnodeRearAxisY.commandConfiguration.camIn.applicationMode := 0;
   cmMendrelAnodeRearAxisY.commandConfiguration.camIn.syncDirection := 1;
   cmMendrelAnodeRearAxisY.commandConfiguration.gearOutCamOut.slavePosition := 0.0;
   cmMendrelAnodeRearAxisY.commandConfiguration.gearOutCamOut.syncProfileReference := 1;
   cmMendrelAnodeRearAxisY.commandConfiguration.gearOutCamOut.masterStopDistance := 0.0;
   cmMendrelAnodeRearAxisY.commandConfiguration.gearOutCamOut.deceleration := -1.0;
   cmMendrelAnodeRearAxisY.commandConfiguration.gearOutCamOut.jerk := -1.0;
   cmMendrelAnodeRearAxisY.commandConfiguration.gearOutCamOut.syncOutDirection := 3;
   cmMendrelAnodeRearAxisY.commandConfiguration.gearOutCamOut.gearOutCamOutMode := -1;
   cmMendrelAnodeRearAxisY.commandConfiguration.phasing.phaseShift := 0.0;
   cmMendrelAnodeRearAxisY.commandConfiguration.phasing.velocity := -1.0;
   cmMendrelAnodeRearAxisY.commandConfiguration.phasing.acceleration := -1.0;
   cmMendrelAnodeRearAxisY.commandConfiguration.phasing.deceleration := -1.0;
   cmMendrelAnodeRearAxisY.commandConfiguration.phasing.jerk := -1.0;
   cmMendrelAnodeRearAxisY.commandConfiguration.phasing.profileReference := 0;
   cmMendrelAnodeRearAxisY.commandConfiguration.phasing.phasingDistance := 0.0;
   cmMendrelAnodeRearAxisY.commandConfiguration.phasing.startPosition := 0.0;
   cmMendrelAnodeRearAxisY.commandConfiguration.phasing.direction := 3;
   cmMendrelAnodeRearAxisY.commandConfiguration.phasing.phaseAbsolute := TRUE;
   cmMendrelAnodeRearAxisY.commandConfiguration.phasing.phaseShiftChangeOnTheFly := FALSE;
   cmMendrelAnodeRearAxisY.commandConfiguration.offset.offset := 0.0;
   cmMendrelAnodeRearAxisY.commandConfiguration.offset.profileReference := 1;
   cmMendrelAnodeRearAxisY.commandConfiguration.offset.offsetDistance := 0.0;
   cmMendrelAnodeRearAxisY.commandConfiguration.offset.startPosition := 0.0;
   cmMendrelAnodeRearAxisY.commandConfiguration.offset.direction := 3;
   cmMendrelAnodeRearAxisY.commandConfiguration.offset.offsetAbsolute := TRUE;
   cmMendrelAnodeRearAxisY.commandConfiguration.offset.offsetChangeOnTheFly := FALSE;
   cmMendrelAnodeRearAxisY.commands.enableMasterControl := TRUE;
   cmMendrelAnodeRearAxisY.commands.enableAxis := FALSE;
   cmMendrelAnodeRearAxisY.commands.resetAxis := FALSE;
   cmMendrelAnodeRearAxisY.commands.openBrake := FALSE;
   cmMendrelAnodeRearAxisY.commands.jogForward := FALSE;
   cmMendrelAnodeRearAxisY.commands.jogBackward := FALSE;
   cmMendrelAnodeRearAxisY.commands.moveVelocity := FALSE;
   cmMendrelAnodeRearAxisY.commands.stop := FALSE;
   cmMendrelAnodeRearAxisY.commands.fastStop := FALSE;
   cmMendrelAnodeRearAxisY.commands.torqueLimiting := FALSE;
   cmMendrelAnodeRearAxisY.commands.homing := FALSE;
   cmMendrelAnodeRearAxisY.commands.posRelative := FALSE;
   cmMendrelAnodeRearAxisY.commands.posAbsolute := FALSE;
   cmMendrelAnodeRearAxisY.commands.posSuperimposed := FALSE;
   cmMendrelAnodeRearAxisY.commands.haltSuperimposed := FALSE;
   cmMendrelAnodeRearAxisY.commands.selectSetPosition := 1;
   cmMendrelAnodeRearAxisY.commands.uploadParameters := FALSE;
   cmMendrelAnodeRearAxisY.commands.refreshConfiguration := FALSE;
   cmMendrelAnodeRearAxisY.commands.editConfiguration := FALSE;
   cmMendrelAnodeRearAxisY.commands.saveConfiguration := FALSE;
   cmMendrelAnodeRearAxisY.commands.uploadCurrentTorque := FALSE;
   cmMendrelAnodeRearAxisY.commands.reset := FALSE;
   cmMendrelAnodeRearAxisY.monitoring.enable := TRUE;
   cmMendrelAnodeRearAxisY.monitoring.referenceDesignator := WSTRING#'MendrelAnodeRearAxisY';
   cmMendrelAnodeRearAxisY.monitoring.enabled := TRUE;
   cmMendrelAnodeRearAxisY.monitoring.enableManualCmds := FALSE;
   cmMendrelAnodeRearAxisY.monitoring.reset := FALSE;
   cmMendrelAnodeRearAxisY.monitoring.resetAxis := FALSE;
   cmMendrelAnodeRearAxisY.monitoring.enableAxis := TRUE;
   cmMendrelAnodeRearAxisY.monitoring.openBrake := FALSE;
   cmMendrelAnodeRearAxisY.monitoring.jogBackward := FALSE;
   cmMendrelAnodeRearAxisY.monitoring.jogForward := FALSE;
   cmMendrelAnodeRearAxisY.monitoring.moveVelocity := FALSE;
   cmMendrelAnodeRearAxisY.monitoring.stop := FALSE;
   cmMendrelAnodeRearAxisY.monitoring.fastStop := FALSE;
   cmMendrelAnodeRearAxisY.monitoring.torqueLimiting := FALSE;
   cmMendrelAnodeRearAxisY.monitoring.homing := FALSE;
   cmMendrelAnodeRearAxisY.monitoring.posRelative := FALSE;
   cmMendrelAnodeRearAxisY.monitoring.posAbsolute := FALSE;
   cmMendrelAnodeRearAxisY.monitoring.posSuperimposed := FALSE;
   cmMendrelAnodeRearAxisY.monitoring.haltSuperimposed := FALSE;
   cmMendrelAnodeRearAxisY.monitoring.brakeOpened := FALSE;
   cmMendrelAnodeRearAxisY.monitoring.axisEnabled := TRUE;
   cmMendrelAnodeRearAxisY.monitoring.resetActive := FALSE;
   cmMendrelAnodeRearAxisY.monitoring.inVelocity := FALSE;
   cmMendrelAnodeRearAxisY.monitoring.inLimitation := FALSE;
   cmMendrelAnodeRearAxisY.monitoring.inClamping := FALSE;
   cmMendrelAnodeRearAxisY.monitoring.startSync := FALSE;
   cmMendrelAnodeRearAxisY.monitoring.inSync := FALSE;
   cmMendrelAnodeRearAxisY.monitoring.inSimulation := FALSE;
   cmMendrelAnodeRearAxisY.monitoring.jogSelected := FALSE;
   cmMendrelAnodeRearAxisY.monitoring.moveVelocitySelected := FALSE;
   cmMendrelAnodeRearAxisY.monitoring.stopSelected := FALSE;
   cmMendrelAnodeRearAxisY.monitoring.fastStopSelected := FALSE;
   cmMendrelAnodeRearAxisY.monitoring.torqueLimitingSelected := FALSE;
   cmMendrelAnodeRearAxisY.monitoring.homingSelected := FALSE;
   cmMendrelAnodeRearAxisY.monitoring.posRelativeSelected := FALSE;
   cmMendrelAnodeRearAxisY.monitoring.posAbsoluteSelected := FALSE;
   cmMendrelAnodeRearAxisY.monitoring.posSuperimposedSelected := FALSE;
   cmMendrelAnodeRearAxisY.monitoring.haltSuperimposedSelected := FALSE;
   cmMendrelAnodeRearAxisY.monitoring.commandBusy := FALSE;
   cmMendrelAnodeRearAxisY.monitoring.commandDone := FALSE;
   cmMendrelAnodeRearAxisY.monitoring.commandAborted := FALSE;
   cmMendrelAnodeRearAxisY.monitoring.homingCommandBusy := FALSE;
   cmMendrelAnodeRearAxisY.monitoring.homingCommandDone := FALSE;
   cmMendrelAnodeRearAxisY.monitoring.homingCommandAborted := FALSE;
   cmMendrelAnodeRearAxisY.monitoring.superimposedBusy := FALSE;
   cmMendrelAnodeRearAxisY.monitoring.superimposedDone := FALSE;
   cmMendrelAnodeRearAxisY.monitoring.superimposedAborted := FALSE;
   cmMendrelAnodeRearAxisY.monitoring.selectSetPosition := 1;
   cmMendrelAnodeRearAxisY.monitoring.selectionController := FALSE;
   cmMendrelAnodeRearAxisY.monitoring.interlockGeneral := TRUE;
   cmMendrelAnodeRearAxisY.monitoring.interlockJogForward := TRUE;
   cmMendrelAnodeRearAxisY.monitoring.interlockJogBackward := TRUE;
   cmMendrelAnodeRearAxisY.monitoring.interlockWarningGeneral := FALSE;
   cmMendrelAnodeRearAxisY.monitoring.interlockWarningJogForward := FALSE;
   cmMendrelAnodeRearAxisY.monitoring.interlockWarningJogBackward := FALSE;
   cmMendrelAnodeRearAxisY.monitoring.valid := TRUE;
   cmMendrelAnodeRearAxisY.monitoring.busy := TRUE;
   cmMendrelAnodeRearAxisY.monitoring.error := FALSE;
   cmMendrelAnodeRearAxisY.monitoring.status := 16#7002;
   cmMendrelAnodeRearAxisY.monitoring.subfunctionStatus := 16#0000;
   cmMendrelAnodeRearAxisY.monitoring.actualPosition := 50.0;
   cmMendrelAnodeRearAxisY.monitoring.actualSpeed := 0.0;
   cmMendrelAnodeRearAxisY.monitoring.speedUnit := 1062;
   cmMendrelAnodeRearAxisY.monitoring.positionUnit := 1013;
   cmMendrelAnodeRearAxisY.monitoring.axisStatus1 := 16#0240_10A1;
   cmMendrelAnodeRearAxisY.monitoring.axisStatus2 := 16#0000_0000;
   cmMendrelAnodeRearAxisY.monitoring.axisType := 1;
   cmMendrelAnodeRearAxisY.monitoring.maxVelocity := 2500.0;
   cmMendrelAnodeRearAxisY.monitoring.actualCurrent := 0.0;
   cmMendrelAnodeRearAxisY.monitoring.actualTorque := 0.0;
   cmMendrelAnodeRearAxisY.monitoring.velocityOverrideEnabled := FALSE;
   cmMendrelAnodeRearAxisY.monitoring.sinaParaError := FALSE;
   cmMendrelAnodeRearAxisY.monitoring.sinaParaStatus := 16#0000_0000;
   cmMendrelAnodeRearAxisY.configuration.referenceDesignator := WSTRING#'MendrelAnodeRearAxisY';
   cmMendrelAnodeRearAxisY.configuration.disableAlarms := FALSE;
   cmMendrelAnodeRearAxisY.configuration.masterControlPopUp := TRUE;
   cmMendrelAnodeRearAxisY.configuration.setPositions[0].position := 0.0;
   cmMendrelAnodeRearAxisY.configuration.setPositions[1].position := 50.0;
   cmMendrelAnodeRearAxisY.configuration.setPositions[2..15].position := 0.0;
   cmMendrelAnodeRearAxisY.configuration.setPositions[0..1].velocity := 50.0;
   cmMendrelAnodeRearAxisY.configuration.setPositions[2..15].velocity := -1.0;
   cmMendrelAnodeRearAxisY.configuration.setPositions[0..1].acceleration := 500.0;
   cmMendrelAnodeRearAxisY.configuration.setPositions[2..15].acceleration := -1.0;
   cmMendrelAnodeRearAxisY.configuration.setPositions[0..1].deceleration := 500.0;
   cmMendrelAnodeRearAxisY.configuration.setPositions[2..15].deceleration := -1.0;
   cmMendrelAnodeRearAxisY.configuration.setPositions[0..15]."name" := '';
   cmMendrelAnodeRearAxisZ.commandConfiguration.generalSettings.stopOnError := TRUE;
   cmMendrelAnodeRearAxisZ.commandConfiguration.generalSettings.resetWithRestart := FALSE;
   cmMendrelAnodeRearAxisZ.commandConfiguration.generalSettings.abortWaitingSyncCmd := TRUE;
   cmMendrelAnodeRearAxisZ.commandConfiguration.power.startMode := 1;
   cmMendrelAnodeRearAxisZ.commandConfiguration.power.stopMode := 0;
   cmMendrelAnodeRearAxisZ.commandConfiguration.power.syncMotionSimulation := FALSE;
   cmMendrelAnodeRearAxisZ.commandConfiguration.power.syncMotionSimulationExtendedMode := -1;
   cmMendrelAnodeRearAxisZ.commandConfiguration.jog.velocity := 0.0;
   cmMendrelAnodeRearAxisZ.commandConfiguration.jog.acceleration := -1.0;
   cmMendrelAnodeRearAxisZ.commandConfiguration.jog.deceleration := -1.0;
   cmMendrelAnodeRearAxisZ.commandConfiguration.jog.jerk := -1.0;
   cmMendrelAnodeRearAxisZ.commandConfiguration.jog.positionControlled := TRUE;
   cmMendrelAnodeRearAxisZ.commandConfiguration.jog.increment := 0.0;
   cmMendrelAnodeRearAxisZ.commandConfiguration.jog.mode := 0;
   cmMendrelAnodeRearAxisZ.commandConfiguration.moveVelocity.velocity := 0.0;
   cmMendrelAnodeRearAxisZ.commandConfiguration.moveVelocity.acceleration := -1.0;
   cmMendrelAnodeRearAxisZ.commandConfiguration.moveVelocity.deceleration := -1.0;
   cmMendrelAnodeRearAxisZ.commandConfiguration.moveVelocity.jerk := -1.0;
   cmMendrelAnodeRearAxisZ.commandConfiguration.moveVelocity.direction := 0;
   cmMendrelAnodeRearAxisZ.commandConfiguration.moveVelocity.positionControlled := TRUE;
   cmMendrelAnodeRearAxisZ.commandConfiguration.moveVelocity.velocityChangeOnTheFly := FALSE;
   cmMendrelAnodeRearAxisZ.commandConfiguration.stop.deceleration := -1.0;
   cmMendrelAnodeRearAxisZ.commandConfiguration.stop.jerk := -1.0;
   cmMendrelAnodeRearAxisZ.commandConfiguration.stop.abortAcceleration := FALSE;
   cmMendrelAnodeRearAxisZ.commandConfiguration.fastStop.deceleration := -1.0;
   cmMendrelAnodeRearAxisZ.commandConfiguration.fastStop.jerk := -1.0;
   cmMendrelAnodeRearAxisZ.commandConfiguration.fastStop.abortAcceleration := FALSE;
   cmMendrelAnodeRearAxisZ.commandConfiguration.fastStop.replaceStopPossible := FALSE;
   cmMendrelAnodeRearAxisZ.commandConfiguration.torqueLimiting.limit := -1.0;
   cmMendrelAnodeRearAxisZ.commandConfiguration.torqueLimiting.mode := 0;
   cmMendrelAnodeRearAxisZ.commandConfiguration.homing.position := 0.0;
   cmMendrelAnodeRearAxisZ.commandConfiguration.homing.mode := 0;
   cmMendrelAnodeRearAxisZ.commandConfiguration.homing.sensor := 0;
   cmMendrelAnodeRearAxisZ.commandConfiguration.homing.extendedMode := -1;
   cmMendrelAnodeRearAxisZ.commandConfiguration.homing.extendedModeTorqueLimit := 0.0;
   cmMendrelAnodeRearAxisZ.commandConfiguration.homing.extendedModeTargetPosition := 0.0;
   cmMendrelAnodeRearAxisZ.commandConfiguration.posRelative.distance := 0.0;
   cmMendrelAnodeRearAxisZ.commandConfiguration.posRelative.velocity := -1.0;
   cmMendrelAnodeRearAxisZ.commandConfiguration.posRelative.acceleration := -1.0;
   cmMendrelAnodeRearAxisZ.commandConfiguration.posRelative.deceleration := -1.0;
   cmMendrelAnodeRearAxisZ.commandConfiguration.posRelative.jerk := -1.0;
   cmMendrelAnodeRearAxisZ.commandConfiguration.posRelative.direction := 0;
   cmMendrelAnodeRearAxisZ.commandConfiguration.posAbsolute.position := 0.0;
   cmMendrelAnodeRearAxisZ.commandConfiguration.posAbsolute.velocity := -1.0;
   cmMendrelAnodeRearAxisZ.commandConfiguration.posAbsolute.acceleration := -1.0;
   cmMendrelAnodeRearAxisZ.commandConfiguration.posAbsolute.deceleration := -1.0;
   cmMendrelAnodeRearAxisZ.commandConfiguration.posAbsolute.jerk := -1.0;
   cmMendrelAnodeRearAxisZ.commandConfiguration.posAbsolute.direction := 1;
   cmMendrelAnodeRearAxisZ.commandConfiguration.posAbsolute.positionChangeOnTheFly := FALSE;
   cmMendrelAnodeRearAxisZ.commandConfiguration.posAbsolute.velocityChangeOnTheFly := FALSE;
   cmMendrelAnodeRearAxisZ.commandConfiguration.posSuperimposed.distance := 0.0;
   cmMendrelAnodeRearAxisZ.commandConfiguration.posSuperimposed.velocityDiff := -1.0;
   cmMendrelAnodeRearAxisZ.commandConfiguration.posSuperimposed.acceleration := -1.0;
   cmMendrelAnodeRearAxisZ.commandConfiguration.posSuperimposed.deceleration := -1.0;
   cmMendrelAnodeRearAxisZ.commandConfiguration.posSuperimposed.jerk := -1.0;
   cmMendrelAnodeRearAxisZ.commandConfiguration.posSuperimposed.direction := 0;
   cmMendrelAnodeRearAxisZ.commandConfiguration.haltSuperimposed.deceleration := -1.0;
   cmMendrelAnodeRearAxisZ.commandConfiguration.haltSuperimposed.jerk := -1.0;
   cmMendrelAnodeRearAxisZ.commandConfiguration.haltSuperimposed.abortAcceleration := FALSE;
   cmMendrelAnodeRearAxisZ.commandConfiguration.gearInRelative.ratioNumerator := 1;
   cmMendrelAnodeRearAxisZ.commandConfiguration.gearInRelative.ratioDenominator := 1;
   cmMendrelAnodeRearAxisZ.commandConfiguration.gearInRelative.acceleration := -1.0;
   cmMendrelAnodeRearAxisZ.commandConfiguration.gearInRelative.deceleration := -1.0;
   cmMendrelAnodeRearAxisZ.commandConfiguration.gearInRelative.jerk := -1.0;
   cmMendrelAnodeRearAxisZ.commandConfiguration.gearInRelative.ratioChangeOnTheFly := FALSE;
   cmMendrelAnodeRearAxisZ.commandConfiguration.gearInAbsolute.ratioNumerator := 1;
   cmMendrelAnodeRearAxisZ.commandConfiguration.gearInAbsolute.ratioDenominator := 1;
   cmMendrelAnodeRearAxisZ.commandConfiguration.gearInAbsolute.masterSyncPosition := 0.0;
   cmMendrelAnodeRearAxisZ.commandConfiguration.gearInAbsolute.slaveSyncPosition := 0.0;
   cmMendrelAnodeRearAxisZ.commandConfiguration.gearInAbsolute.syncProfileReference := 1;
   cmMendrelAnodeRearAxisZ.commandConfiguration.gearInAbsolute.masterStartDistance := 0.0;
   cmMendrelAnodeRearAxisZ.commandConfiguration.gearInAbsolute.velocity := -1.0;
   cmMendrelAnodeRearAxisZ.commandConfiguration.gearInAbsolute.acceleration := -1.0;
   cmMendrelAnodeRearAxisZ.commandConfiguration.gearInAbsolute.deceleration := -1.0;
   cmMendrelAnodeRearAxisZ.commandConfiguration.gearInAbsolute.jerk := -1.0;
   cmMendrelAnodeRearAxisZ.commandConfiguration.gearInAbsolute.syncDirection := 1;
   cmMendrelAnodeRearAxisZ.commandConfiguration.gearInAbsolute.ratioChangeOnTheFly := FALSE;
   cmMendrelAnodeRearAxisZ.commandConfiguration.gearInVelocity.continuousUpdate := FALSE;
   cmMendrelAnodeRearAxisZ.commandConfiguration.gearInVelocity.ratioNumerator := 1;
   cmMendrelAnodeRearAxisZ.commandConfiguration.gearInVelocity.ratioDenominator := 1;
   cmMendrelAnodeRearAxisZ.commandConfiguration.gearInVelocity.acceleration := -1.0;
   cmMendrelAnodeRearAxisZ.commandConfiguration.gearInVelocity.deceleration := -1.0;
   cmMendrelAnodeRearAxisZ.commandConfiguration.gearInVelocity.jerk := -1.0;
   cmMendrelAnodeRearAxisZ.commandConfiguration.gearInVelocity.positionControlled := FALSE;
   cmMendrelAnodeRearAxisZ.commandConfiguration.camIn.masterOffset := 0.0;
   cmMendrelAnodeRearAxisZ.commandConfiguration.camIn.slaveOffset := 0.0;
   cmMendrelAnodeRearAxisZ.commandConfiguration.camIn.masterScaling := 1.0;
   cmMendrelAnodeRearAxisZ.commandConfiguration.camIn.slaveScaling := 1.0;
   cmMendrelAnodeRearAxisZ.commandConfiguration.camIn.masterSyncPosition := 0.0;
   cmMendrelAnodeRearAxisZ.commandConfiguration.camIn.syncProfileReference := 1;
   cmMendrelAnodeRearAxisZ.commandConfiguration.camIn.masterStartDistance := 0.0;
   cmMendrelAnodeRearAxisZ.commandConfiguration.camIn.velocity := -1.0;
   cmMendrelAnodeRearAxisZ.commandConfiguration.camIn.acceleration := -1.0;
   cmMendrelAnodeRearAxisZ.commandConfiguration.camIn.deceleration := -1.0;
   cmMendrelAnodeRearAxisZ.commandConfiguration.camIn.jerk := -1.0;
   cmMendrelAnodeRearAxisZ.commandConfiguration.camIn.applicationMode := 0;
   cmMendrelAnodeRearAxisZ.commandConfiguration.camIn.syncDirection := 1;
   cmMendrelAnodeRearAxisZ.commandConfiguration.gearOutCamOut.slavePosition := 0.0;
   cmMendrelAnodeRearAxisZ.commandConfiguration.gearOutCamOut.syncProfileReference := 1;
   cmMendrelAnodeRearAxisZ.commandConfiguration.gearOutCamOut.masterStopDistance := 0.0;
   cmMendrelAnodeRearAxisZ.commandConfiguration.gearOutCamOut.deceleration := -1.0;
   cmMendrelAnodeRearAxisZ.commandConfiguration.gearOutCamOut.jerk := -1.0;
   cmMendrelAnodeRearAxisZ.commandConfiguration.gearOutCamOut.syncOutDirection := 3;
   cmMendrelAnodeRearAxisZ.commandConfiguration.gearOutCamOut.gearOutCamOutMode := -1;
   cmMendrelAnodeRearAxisZ.commandConfiguration.phasing.phaseShift := 0.0;
   cmMendrelAnodeRearAxisZ.commandConfiguration.phasing.velocity := -1.0;
   cmMendrelAnodeRearAxisZ.commandConfiguration.phasing.acceleration := -1.0;
   cmMendrelAnodeRearAxisZ.commandConfiguration.phasing.deceleration := -1.0;
   cmMendrelAnodeRearAxisZ.commandConfiguration.phasing.jerk := -1.0;
   cmMendrelAnodeRearAxisZ.commandConfiguration.phasing.profileReference := 0;
   cmMendrelAnodeRearAxisZ.commandConfiguration.phasing.phasingDistance := 0.0;
   cmMendrelAnodeRearAxisZ.commandConfiguration.phasing.startPosition := 0.0;
   cmMendrelAnodeRearAxisZ.commandConfiguration.phasing.direction := 3;
   cmMendrelAnodeRearAxisZ.commandConfiguration.phasing.phaseAbsolute := TRUE;
   cmMendrelAnodeRearAxisZ.commandConfiguration.phasing.phaseShiftChangeOnTheFly := FALSE;
   cmMendrelAnodeRearAxisZ.commandConfiguration.offset.offset := 0.0;
   cmMendrelAnodeRearAxisZ.commandConfiguration.offset.profileReference := 1;
   cmMendrelAnodeRearAxisZ.commandConfiguration.offset.offsetDistance := 0.0;
   cmMendrelAnodeRearAxisZ.commandConfiguration.offset.startPosition := 0.0;
   cmMendrelAnodeRearAxisZ.commandConfiguration.offset.direction := 3;
   cmMendrelAnodeRearAxisZ.commandConfiguration.offset.offsetAbsolute := TRUE;
   cmMendrelAnodeRearAxisZ.commandConfiguration.offset.offsetChangeOnTheFly := FALSE;
   cmMendrelAnodeRearAxisZ.commands.enableMasterControl := TRUE;
   cmMendrelAnodeRearAxisZ.commands.enableAxis := FALSE;
   cmMendrelAnodeRearAxisZ.commands.resetAxis := FALSE;
   cmMendrelAnodeRearAxisZ.commands.openBrake := FALSE;
   cmMendrelAnodeRearAxisZ.commands.jogForward := FALSE;
   cmMendrelAnodeRearAxisZ.commands.jogBackward := FALSE;
   cmMendrelAnodeRearAxisZ.commands.moveVelocity := FALSE;
   cmMendrelAnodeRearAxisZ.commands.stop := FALSE;
   cmMendrelAnodeRearAxisZ.commands.fastStop := FALSE;
   cmMendrelAnodeRearAxisZ.commands.torqueLimiting := FALSE;
   cmMendrelAnodeRearAxisZ.commands.homing := FALSE;
   cmMendrelAnodeRearAxisZ.commands.posRelative := FALSE;
   cmMendrelAnodeRearAxisZ.commands.posAbsolute := FALSE;
   cmMendrelAnodeRearAxisZ.commands.posSuperimposed := FALSE;
   cmMendrelAnodeRearAxisZ.commands.haltSuperimposed := FALSE;
   cmMendrelAnodeRearAxisZ.commands.selectSetPosition := 1;
   cmMendrelAnodeRearAxisZ.commands.uploadParameters := FALSE;
   cmMendrelAnodeRearAxisZ.commands.refreshConfiguration := FALSE;
   cmMendrelAnodeRearAxisZ.commands.editConfiguration := FALSE;
   cmMendrelAnodeRearAxisZ.commands.saveConfiguration := FALSE;
   cmMendrelAnodeRearAxisZ.commands.uploadCurrentTorque := FALSE;
   cmMendrelAnodeRearAxisZ.commands.reset := FALSE;
   cmMendrelAnodeRearAxisZ.monitoring.enable := TRUE;
   cmMendrelAnodeRearAxisZ.monitoring.referenceDesignator := WSTRING#'MendrelAnodeRearAxisZ';
   cmMendrelAnodeRearAxisZ.monitoring.enabled := TRUE;
   cmMendrelAnodeRearAxisZ.monitoring.enableManualCmds := FALSE;
   cmMendrelAnodeRearAxisZ.monitoring.reset := FALSE;
   cmMendrelAnodeRearAxisZ.monitoring.resetAxis := FALSE;
   cmMendrelAnodeRearAxisZ.monitoring.enableAxis := TRUE;
   cmMendrelAnodeRearAxisZ.monitoring.openBrake := FALSE;
   cmMendrelAnodeRearAxisZ.monitoring.jogBackward := FALSE;
   cmMendrelAnodeRearAxisZ.monitoring.jogForward := FALSE;
   cmMendrelAnodeRearAxisZ.monitoring.moveVelocity := FALSE;
   cmMendrelAnodeRearAxisZ.monitoring.stop := FALSE;
   cmMendrelAnodeRearAxisZ.monitoring.fastStop := FALSE;
   cmMendrelAnodeRearAxisZ.monitoring.torqueLimiting := FALSE;
   cmMendrelAnodeRearAxisZ.monitoring.homing := FALSE;
   cmMendrelAnodeRearAxisZ.monitoring.posRelative := FALSE;
   cmMendrelAnodeRearAxisZ.monitoring.posAbsolute := FALSE;
   cmMendrelAnodeRearAxisZ.monitoring.posSuperimposed := FALSE;
   cmMendrelAnodeRearAxisZ.monitoring.haltSuperimposed := FALSE;
   cmMendrelAnodeRearAxisZ.monitoring.brakeOpened := FALSE;
   cmMendrelAnodeRearAxisZ.monitoring.axisEnabled := TRUE;
   cmMendrelAnodeRearAxisZ.monitoring.resetActive := FALSE;
   cmMendrelAnodeRearAxisZ.monitoring.inVelocity := FALSE;
   cmMendrelAnodeRearAxisZ.monitoring.inLimitation := FALSE;
   cmMendrelAnodeRearAxisZ.monitoring.inClamping := FALSE;
   cmMendrelAnodeRearAxisZ.monitoring.startSync := FALSE;
   cmMendrelAnodeRearAxisZ.monitoring.inSync := FALSE;
   cmMendrelAnodeRearAxisZ.monitoring.inSimulation := FALSE;
   cmMendrelAnodeRearAxisZ.monitoring.jogSelected := FALSE;
   cmMendrelAnodeRearAxisZ.monitoring.moveVelocitySelected := FALSE;
   cmMendrelAnodeRearAxisZ.monitoring.stopSelected := FALSE;
   cmMendrelAnodeRearAxisZ.monitoring.fastStopSelected := FALSE;
   cmMendrelAnodeRearAxisZ.monitoring.torqueLimitingSelected := FALSE;
   cmMendrelAnodeRearAxisZ.monitoring.homingSelected := FALSE;
   cmMendrelAnodeRearAxisZ.monitoring.posRelativeSelected := FALSE;
   cmMendrelAnodeRearAxisZ.monitoring.posAbsoluteSelected := FALSE;
   cmMendrelAnodeRearAxisZ.monitoring.posSuperimposedSelected := FALSE;
   cmMendrelAnodeRearAxisZ.monitoring.haltSuperimposedSelected := FALSE;
   cmMendrelAnodeRearAxisZ.monitoring.commandBusy := FALSE;
   cmMendrelAnodeRearAxisZ.monitoring.commandDone := FALSE;
   cmMendrelAnodeRearAxisZ.monitoring.commandAborted := FALSE;
   cmMendrelAnodeRearAxisZ.monitoring.homingCommandBusy := FALSE;
   cmMendrelAnodeRearAxisZ.monitoring.homingCommandDone := FALSE;
   cmMendrelAnodeRearAxisZ.monitoring.homingCommandAborted := FALSE;
   cmMendrelAnodeRearAxisZ.monitoring.superimposedBusy := FALSE;
   cmMendrelAnodeRearAxisZ.monitoring.superimposedDone := FALSE;
   cmMendrelAnodeRearAxisZ.monitoring.superimposedAborted := FALSE;
   cmMendrelAnodeRearAxisZ.monitoring.selectSetPosition := 1;
   cmMendrelAnodeRearAxisZ.monitoring.selectionController := FALSE;
   cmMendrelAnodeRearAxisZ.monitoring.interlockGeneral := TRUE;
   cmMendrelAnodeRearAxisZ.monitoring.interlockJogForward := TRUE;
   cmMendrelAnodeRearAxisZ.monitoring.interlockJogBackward := TRUE;
   cmMendrelAnodeRearAxisZ.monitoring.interlockWarningGeneral := FALSE;
   cmMendrelAnodeRearAxisZ.monitoring.interlockWarningJogForward := FALSE;
   cmMendrelAnodeRearAxisZ.monitoring.interlockWarningJogBackward := FALSE;
   cmMendrelAnodeRearAxisZ.monitoring.valid := TRUE;
   cmMendrelAnodeRearAxisZ.monitoring.busy := TRUE;
   cmMendrelAnodeRearAxisZ.monitoring.error := FALSE;
   cmMendrelAnodeRearAxisZ.monitoring.status := 16#7002;
   cmMendrelAnodeRearAxisZ.monitoring.subfunctionStatus := 16#0000;
   cmMendrelAnodeRearAxisZ.monitoring.actualPosition := 50.0;
   cmMendrelAnodeRearAxisZ.monitoring.actualSpeed := 0.0;
   cmMendrelAnodeRearAxisZ.monitoring.speedUnit := 1062;
   cmMendrelAnodeRearAxisZ.monitoring.positionUnit := 1013;
   cmMendrelAnodeRearAxisZ.monitoring.axisStatus1 := 16#0240_10A1;
   cmMendrelAnodeRearAxisZ.monitoring.axisStatus2 := 16#0000_0000;
   cmMendrelAnodeRearAxisZ.monitoring.axisType := 1;
   cmMendrelAnodeRearAxisZ.monitoring.maxVelocity := 2500.0;
   cmMendrelAnodeRearAxisZ.monitoring.actualCurrent := 0.0;
   cmMendrelAnodeRearAxisZ.monitoring.actualTorque := 0.0;
   cmMendrelAnodeRearAxisZ.monitoring.velocityOverrideEnabled := FALSE;
   cmMendrelAnodeRearAxisZ.monitoring.sinaParaError := FALSE;
   cmMendrelAnodeRearAxisZ.monitoring.sinaParaStatus := 16#0000_0000;
   cmMendrelAnodeRearAxisZ.configuration.referenceDesignator := WSTRING#'MendrelAnodeRearAxisZ';
   cmMendrelAnodeRearAxisZ.configuration.disableAlarms := FALSE;
   cmMendrelAnodeRearAxisZ.configuration.masterControlPopUp := TRUE;
   cmMendrelAnodeRearAxisZ.configuration.setPositions[0].position := 0.0;
   cmMendrelAnodeRearAxisZ.configuration.setPositions[1].position := 50.0;
   cmMendrelAnodeRearAxisZ.configuration.setPositions[2..15].position := 0.0;
   cmMendrelAnodeRearAxisZ.configuration.setPositions[0..1].velocity := 50.0;
   cmMendrelAnodeRearAxisZ.configuration.setPositions[2..15].velocity := -1.0;
   cmMendrelAnodeRearAxisZ.configuration.setPositions[0..1].acceleration := 500.0;
   cmMendrelAnodeRearAxisZ.configuration.setPositions[2..15].acceleration := -1.0;
   cmMendrelAnodeRearAxisZ.configuration.setPositions[0..1].deceleration := 500.0;
   cmMendrelAnodeRearAxisZ.configuration.setPositions[2..15].deceleration := -1.0;
   cmMendrelAnodeRearAxisZ.configuration.setPositions[0..15]."name" := '';
   cmMendrelCathodeFrontAxisY.commandConfiguration.generalSettings.stopOnError := TRUE;
   cmMendrelCathodeFrontAxisY.commandConfiguration.generalSettings.resetWithRestart := FALSE;
   cmMendrelCathodeFrontAxisY.commandConfiguration.generalSettings.abortWaitingSyncCmd := TRUE;
   cmMendrelCathodeFrontAxisY.commandConfiguration.power.startMode := 1;
   cmMendrelCathodeFrontAxisY.commandConfiguration.power.stopMode := 0;
   cmMendrelCathodeFrontAxisY.commandConfiguration.power.syncMotionSimulation := FALSE;
   cmMendrelCathodeFrontAxisY.commandConfiguration.power.syncMotionSimulationExtendedMode := -1;
   cmMendrelCathodeFrontAxisY.commandConfiguration.jog.velocity := 0.0;
   cmMendrelCathodeFrontAxisY.commandConfiguration.jog.acceleration := -1.0;
   cmMendrelCathodeFrontAxisY.commandConfiguration.jog.deceleration := -1.0;
   cmMendrelCathodeFrontAxisY.commandConfiguration.jog.jerk := -1.0;
   cmMendrelCathodeFrontAxisY.commandConfiguration.jog.positionControlled := TRUE;
   cmMendrelCathodeFrontAxisY.commandConfiguration.jog.increment := 0.0;
   cmMendrelCathodeFrontAxisY.commandConfiguration.jog.mode := 0;
   cmMendrelCathodeFrontAxisY.commandConfiguration.moveVelocity.velocity := 0.0;
   cmMendrelCathodeFrontAxisY.commandConfiguration.moveVelocity.acceleration := -1.0;
   cmMendrelCathodeFrontAxisY.commandConfiguration.moveVelocity.deceleration := -1.0;
   cmMendrelCathodeFrontAxisY.commandConfiguration.moveVelocity.jerk := -1.0;
   cmMendrelCathodeFrontAxisY.commandConfiguration.moveVelocity.direction := 0;
   cmMendrelCathodeFrontAxisY.commandConfiguration.moveVelocity.positionControlled := TRUE;
   cmMendrelCathodeFrontAxisY.commandConfiguration.moveVelocity.velocityChangeOnTheFly := FALSE;
   cmMendrelCathodeFrontAxisY.commandConfiguration.stop.deceleration := -1.0;
   cmMendrelCathodeFrontAxisY.commandConfiguration.stop.jerk := -1.0;
   cmMendrelCathodeFrontAxisY.commandConfiguration.stop.abortAcceleration := FALSE;
   cmMendrelCathodeFrontAxisY.commandConfiguration.fastStop.deceleration := -1.0;
   cmMendrelCathodeFrontAxisY.commandConfiguration.fastStop.jerk := -1.0;
   cmMendrelCathodeFrontAxisY.commandConfiguration.fastStop.abortAcceleration := FALSE;
   cmMendrelCathodeFrontAxisY.commandConfiguration.fastStop.replaceStopPossible := FALSE;
   cmMendrelCathodeFrontAxisY.commandConfiguration.torqueLimiting.limit := -1.0;
   cmMendrelCathodeFrontAxisY.commandConfiguration.torqueLimiting.mode := 0;
   cmMendrelCathodeFrontAxisY.commandConfiguration.homing.position := 0.0;
   cmMendrelCathodeFrontAxisY.commandConfiguration.homing.mode := 0;
   cmMendrelCathodeFrontAxisY.commandConfiguration.homing.sensor := 0;
   cmMendrelCathodeFrontAxisY.commandConfiguration.homing.extendedMode := -1;
   cmMendrelCathodeFrontAxisY.commandConfiguration.homing.extendedModeTorqueLimit := 0.0;
   cmMendrelCathodeFrontAxisY.commandConfiguration.homing.extendedModeTargetPosition := 0.0;
   cmMendrelCathodeFrontAxisY.commandConfiguration.posRelative.distance := 0.0;
   cmMendrelCathodeFrontAxisY.commandConfiguration.posRelative.velocity := -1.0;
   cmMendrelCathodeFrontAxisY.commandConfiguration.posRelative.acceleration := -1.0;
   cmMendrelCathodeFrontAxisY.commandConfiguration.posRelative.deceleration := -1.0;
   cmMendrelCathodeFrontAxisY.commandConfiguration.posRelative.jerk := -1.0;
   cmMendrelCathodeFrontAxisY.commandConfiguration.posRelative.direction := 0;
   cmMendrelCathodeFrontAxisY.commandConfiguration.posAbsolute.position := 0.0;
   cmMendrelCathodeFrontAxisY.commandConfiguration.posAbsolute.velocity := -1.0;
   cmMendrelCathodeFrontAxisY.commandConfiguration.posAbsolute.acceleration := -1.0;
   cmMendrelCathodeFrontAxisY.commandConfiguration.posAbsolute.deceleration := -1.0;
   cmMendrelCathodeFrontAxisY.commandConfiguration.posAbsolute.jerk := -1.0;
   cmMendrelCathodeFrontAxisY.commandConfiguration.posAbsolute.direction := 1;
   cmMendrelCathodeFrontAxisY.commandConfiguration.posAbsolute.positionChangeOnTheFly := FALSE;
   cmMendrelCathodeFrontAxisY.commandConfiguration.posAbsolute.velocityChangeOnTheFly := FALSE;
   cmMendrelCathodeFrontAxisY.commandConfiguration.posSuperimposed.distance := 0.0;
   cmMendrelCathodeFrontAxisY.commandConfiguration.posSuperimposed.velocityDiff := -1.0;
   cmMendrelCathodeFrontAxisY.commandConfiguration.posSuperimposed.acceleration := -1.0;
   cmMendrelCathodeFrontAxisY.commandConfiguration.posSuperimposed.deceleration := -1.0;
   cmMendrelCathodeFrontAxisY.commandConfiguration.posSuperimposed.jerk := -1.0;
   cmMendrelCathodeFrontAxisY.commandConfiguration.posSuperimposed.direction := 0;
   cmMendrelCathodeFrontAxisY.commandConfiguration.haltSuperimposed.deceleration := -1.0;
   cmMendrelCathodeFrontAxisY.commandConfiguration.haltSuperimposed.jerk := -1.0;
   cmMendrelCathodeFrontAxisY.commandConfiguration.haltSuperimposed.abortAcceleration := FALSE;
   cmMendrelCathodeFrontAxisY.commandConfiguration.gearInRelative.ratioNumerator := 1;
   cmMendrelCathodeFrontAxisY.commandConfiguration.gearInRelative.ratioDenominator := 1;
   cmMendrelCathodeFrontAxisY.commandConfiguration.gearInRelative.acceleration := -1.0;
   cmMendrelCathodeFrontAxisY.commandConfiguration.gearInRelative.deceleration := -1.0;
   cmMendrelCathodeFrontAxisY.commandConfiguration.gearInRelative.jerk := -1.0;
   cmMendrelCathodeFrontAxisY.commandConfiguration.gearInRelative.ratioChangeOnTheFly := FALSE;
   cmMendrelCathodeFrontAxisY.commandConfiguration.gearInAbsolute.ratioNumerator := 1;
   cmMendrelCathodeFrontAxisY.commandConfiguration.gearInAbsolute.ratioDenominator := 1;
   cmMendrelCathodeFrontAxisY.commandConfiguration.gearInAbsolute.masterSyncPosition := 0.0;
   cmMendrelCathodeFrontAxisY.commandConfiguration.gearInAbsolute.slaveSyncPosition := 0.0;
   cmMendrelCathodeFrontAxisY.commandConfiguration.gearInAbsolute.syncProfileReference := 1;
   cmMendrelCathodeFrontAxisY.commandConfiguration.gearInAbsolute.masterStartDistance := 0.0;
   cmMendrelCathodeFrontAxisY.commandConfiguration.gearInAbsolute.velocity := -1.0;
   cmMendrelCathodeFrontAxisY.commandConfiguration.gearInAbsolute.acceleration := -1.0;
   cmMendrelCathodeFrontAxisY.commandConfiguration.gearInAbsolute.deceleration := -1.0;
   cmMendrelCathodeFrontAxisY.commandConfiguration.gearInAbsolute.jerk := -1.0;
   cmMendrelCathodeFrontAxisY.commandConfiguration.gearInAbsolute.syncDirection := 1;
   cmMendrelCathodeFrontAxisY.commandConfiguration.gearInAbsolute.ratioChangeOnTheFly := FALSE;
   cmMendrelCathodeFrontAxisY.commandConfiguration.gearInVelocity.continuousUpdate := FALSE;
   cmMendrelCathodeFrontAxisY.commandConfiguration.gearInVelocity.ratioNumerator := 1;
   cmMendrelCathodeFrontAxisY.commandConfiguration.gearInVelocity.ratioDenominator := 1;
   cmMendrelCathodeFrontAxisY.commandConfiguration.gearInVelocity.acceleration := -1.0;
   cmMendrelCathodeFrontAxisY.commandConfiguration.gearInVelocity.deceleration := -1.0;
   cmMendrelCathodeFrontAxisY.commandConfiguration.gearInVelocity.jerk := -1.0;
   cmMendrelCathodeFrontAxisY.commandConfiguration.gearInVelocity.positionControlled := FALSE;
   cmMendrelCathodeFrontAxisY.commandConfiguration.camIn.masterOffset := 0.0;
   cmMendrelCathodeFrontAxisY.commandConfiguration.camIn.slaveOffset := 0.0;
   cmMendrelCathodeFrontAxisY.commandConfiguration.camIn.masterScaling := 1.0;
   cmMendrelCathodeFrontAxisY.commandConfiguration.camIn.slaveScaling := 1.0;
   cmMendrelCathodeFrontAxisY.commandConfiguration.camIn.masterSyncPosition := 0.0;
   cmMendrelCathodeFrontAxisY.commandConfiguration.camIn.syncProfileReference := 1;
   cmMendrelCathodeFrontAxisY.commandConfiguration.camIn.masterStartDistance := 0.0;
   cmMendrelCathodeFrontAxisY.commandConfiguration.camIn.velocity := -1.0;
   cmMendrelCathodeFrontAxisY.commandConfiguration.camIn.acceleration := -1.0;
   cmMendrelCathodeFrontAxisY.commandConfiguration.camIn.deceleration := -1.0;
   cmMendrelCathodeFrontAxisY.commandConfiguration.camIn.jerk := -1.0;
   cmMendrelCathodeFrontAxisY.commandConfiguration.camIn.applicationMode := 0;
   cmMendrelCathodeFrontAxisY.commandConfiguration.camIn.syncDirection := 1;
   cmMendrelCathodeFrontAxisY.commandConfiguration.gearOutCamOut.slavePosition := 0.0;
   cmMendrelCathodeFrontAxisY.commandConfiguration.gearOutCamOut.syncProfileReference := 1;
   cmMendrelCathodeFrontAxisY.commandConfiguration.gearOutCamOut.masterStopDistance := 0.0;
   cmMendrelCathodeFrontAxisY.commandConfiguration.gearOutCamOut.deceleration := -1.0;
   cmMendrelCathodeFrontAxisY.commandConfiguration.gearOutCamOut.jerk := -1.0;
   cmMendrelCathodeFrontAxisY.commandConfiguration.gearOutCamOut.syncOutDirection := 3;
   cmMendrelCathodeFrontAxisY.commandConfiguration.gearOutCamOut.gearOutCamOutMode := -1;
   cmMendrelCathodeFrontAxisY.commandConfiguration.phasing.phaseShift := 0.0;
   cmMendrelCathodeFrontAxisY.commandConfiguration.phasing.velocity := -1.0;
   cmMendrelCathodeFrontAxisY.commandConfiguration.phasing.acceleration := -1.0;
   cmMendrelCathodeFrontAxisY.commandConfiguration.phasing.deceleration := -1.0;
   cmMendrelCathodeFrontAxisY.commandConfiguration.phasing.jerk := -1.0;
   cmMendrelCathodeFrontAxisY.commandConfiguration.phasing.profileReference := 0;
   cmMendrelCathodeFrontAxisY.commandConfiguration.phasing.phasingDistance := 0.0;
   cmMendrelCathodeFrontAxisY.commandConfiguration.phasing.startPosition := 0.0;
   cmMendrelCathodeFrontAxisY.commandConfiguration.phasing.direction := 3;
   cmMendrelCathodeFrontAxisY.commandConfiguration.phasing.phaseAbsolute := TRUE;
   cmMendrelCathodeFrontAxisY.commandConfiguration.phasing.phaseShiftChangeOnTheFly := FALSE;
   cmMendrelCathodeFrontAxisY.commandConfiguration.offset.offset := 0.0;
   cmMendrelCathodeFrontAxisY.commandConfiguration.offset.profileReference := 1;
   cmMendrelCathodeFrontAxisY.commandConfiguration.offset.offsetDistance := 0.0;
   cmMendrelCathodeFrontAxisY.commandConfiguration.offset.startPosition := 0.0;
   cmMendrelCathodeFrontAxisY.commandConfiguration.offset.direction := 3;
   cmMendrelCathodeFrontAxisY.commandConfiguration.offset.offsetAbsolute := TRUE;
   cmMendrelCathodeFrontAxisY.commandConfiguration.offset.offsetChangeOnTheFly := FALSE;
   cmMendrelCathodeFrontAxisY.commands.enableMasterControl := TRUE;
   cmMendrelCathodeFrontAxisY.commands.enableAxis := FALSE;
   cmMendrelCathodeFrontAxisY.commands.resetAxis := FALSE;
   cmMendrelCathodeFrontAxisY.commands.openBrake := FALSE;
   cmMendrelCathodeFrontAxisY.commands.jogForward := FALSE;
   cmMendrelCathodeFrontAxisY.commands.jogBackward := FALSE;
   cmMendrelCathodeFrontAxisY.commands.moveVelocity := FALSE;
   cmMendrelCathodeFrontAxisY.commands.stop := FALSE;
   cmMendrelCathodeFrontAxisY.commands.fastStop := FALSE;
   cmMendrelCathodeFrontAxisY.commands.torqueLimiting := FALSE;
   cmMendrelCathodeFrontAxisY.commands.homing := FALSE;
   cmMendrelCathodeFrontAxisY.commands.posRelative := FALSE;
   cmMendrelCathodeFrontAxisY.commands.posAbsolute := FALSE;
   cmMendrelCathodeFrontAxisY.commands.posSuperimposed := FALSE;
   cmMendrelCathodeFrontAxisY.commands.haltSuperimposed := FALSE;
   cmMendrelCathodeFrontAxisY.commands.selectSetPosition := 1;
   cmMendrelCathodeFrontAxisY.commands.uploadParameters := FALSE;
   cmMendrelCathodeFrontAxisY.commands.refreshConfiguration := FALSE;
   cmMendrelCathodeFrontAxisY.commands.editConfiguration := FALSE;
   cmMendrelCathodeFrontAxisY.commands.saveConfiguration := FALSE;
   cmMendrelCathodeFrontAxisY.commands.uploadCurrentTorque := FALSE;
   cmMendrelCathodeFrontAxisY.commands.reset := FALSE;
   cmMendrelCathodeFrontAxisY.monitoring.enable := TRUE;
   cmMendrelCathodeFrontAxisY.monitoring.referenceDesignator := WSTRING#'MendrelCathodeFrontAxisY';
   cmMendrelCathodeFrontAxisY.monitoring.enabled := TRUE;
   cmMendrelCathodeFrontAxisY.monitoring.enableManualCmds := FALSE;
   cmMendrelCathodeFrontAxisY.monitoring.reset := FALSE;
   cmMendrelCathodeFrontAxisY.monitoring.resetAxis := FALSE;
   cmMendrelCathodeFrontAxisY.monitoring.enableAxis := TRUE;
   cmMendrelCathodeFrontAxisY.monitoring.openBrake := FALSE;
   cmMendrelCathodeFrontAxisY.monitoring.jogBackward := FALSE;
   cmMendrelCathodeFrontAxisY.monitoring.jogForward := FALSE;
   cmMendrelCathodeFrontAxisY.monitoring.moveVelocity := FALSE;
   cmMendrelCathodeFrontAxisY.monitoring.stop := FALSE;
   cmMendrelCathodeFrontAxisY.monitoring.fastStop := FALSE;
   cmMendrelCathodeFrontAxisY.monitoring.torqueLimiting := FALSE;
   cmMendrelCathodeFrontAxisY.monitoring.homing := FALSE;
   cmMendrelCathodeFrontAxisY.monitoring.posRelative := FALSE;
   cmMendrelCathodeFrontAxisY.monitoring.posAbsolute := FALSE;
   cmMendrelCathodeFrontAxisY.monitoring.posSuperimposed := FALSE;
   cmMendrelCathodeFrontAxisY.monitoring.haltSuperimposed := FALSE;
   cmMendrelCathodeFrontAxisY.monitoring.brakeOpened := FALSE;
   cmMendrelCathodeFrontAxisY.monitoring.axisEnabled := TRUE;
   cmMendrelCathodeFrontAxisY.monitoring.resetActive := FALSE;
   cmMendrelCathodeFrontAxisY.monitoring.inVelocity := FALSE;
   cmMendrelCathodeFrontAxisY.monitoring.inLimitation := FALSE;
   cmMendrelCathodeFrontAxisY.monitoring.inClamping := FALSE;
   cmMendrelCathodeFrontAxisY.monitoring.startSync := FALSE;
   cmMendrelCathodeFrontAxisY.monitoring.inSync := FALSE;
   cmMendrelCathodeFrontAxisY.monitoring.inSimulation := FALSE;
   cmMendrelCathodeFrontAxisY.monitoring.jogSelected := FALSE;
   cmMendrelCathodeFrontAxisY.monitoring.moveVelocitySelected := FALSE;
   cmMendrelCathodeFrontAxisY.monitoring.stopSelected := FALSE;
   cmMendrelCathodeFrontAxisY.monitoring.fastStopSelected := FALSE;
   cmMendrelCathodeFrontAxisY.monitoring.torqueLimitingSelected := FALSE;
   cmMendrelCathodeFrontAxisY.monitoring.homingSelected := FALSE;
   cmMendrelCathodeFrontAxisY.monitoring.posRelativeSelected := FALSE;
   cmMendrelCathodeFrontAxisY.monitoring.posAbsoluteSelected := FALSE;
   cmMendrelCathodeFrontAxisY.monitoring.posSuperimposedSelected := FALSE;
   cmMendrelCathodeFrontAxisY.monitoring.haltSuperimposedSelected := FALSE;
   cmMendrelCathodeFrontAxisY.monitoring.commandBusy := FALSE;
   cmMendrelCathodeFrontAxisY.monitoring.commandDone := FALSE;
   cmMendrelCathodeFrontAxisY.monitoring.commandAborted := FALSE;
   cmMendrelCathodeFrontAxisY.monitoring.homingCommandBusy := FALSE;
   cmMendrelCathodeFrontAxisY.monitoring.homingCommandDone := FALSE;
   cmMendrelCathodeFrontAxisY.monitoring.homingCommandAborted := FALSE;
   cmMendrelCathodeFrontAxisY.monitoring.superimposedBusy := FALSE;
   cmMendrelCathodeFrontAxisY.monitoring.superimposedDone := FALSE;
   cmMendrelCathodeFrontAxisY.monitoring.superimposedAborted := FALSE;
   cmMendrelCathodeFrontAxisY.monitoring.selectSetPosition := 1;
   cmMendrelCathodeFrontAxisY.monitoring.selectionController := FALSE;
   cmMendrelCathodeFrontAxisY.monitoring.interlockGeneral := TRUE;
   cmMendrelCathodeFrontAxisY.monitoring.interlockJogForward := TRUE;
   cmMendrelCathodeFrontAxisY.monitoring.interlockJogBackward := TRUE;
   cmMendrelCathodeFrontAxisY.monitoring.interlockWarningGeneral := FALSE;
   cmMendrelCathodeFrontAxisY.monitoring.interlockWarningJogForward := FALSE;
   cmMendrelCathodeFrontAxisY.monitoring.interlockWarningJogBackward := FALSE;
   cmMendrelCathodeFrontAxisY.monitoring.valid := TRUE;
   cmMendrelCathodeFrontAxisY.monitoring.busy := TRUE;
   cmMendrelCathodeFrontAxisY.monitoring.error := FALSE;
   cmMendrelCathodeFrontAxisY.monitoring.status := 16#7002;
   cmMendrelCathodeFrontAxisY.monitoring.subfunctionStatus := 16#0000;
   cmMendrelCathodeFrontAxisY.monitoring.actualPosition := 50.0;
   cmMendrelCathodeFrontAxisY.monitoring.actualSpeed := 0.0;
   cmMendrelCathodeFrontAxisY.monitoring.speedUnit := 1062;
   cmMendrelCathodeFrontAxisY.monitoring.positionUnit := 1013;
   cmMendrelCathodeFrontAxisY.monitoring.axisStatus1 := 16#0240_10A1;
   cmMendrelCathodeFrontAxisY.monitoring.axisStatus2 := 16#0000_0000;
   cmMendrelCathodeFrontAxisY.monitoring.axisType := 1;
   cmMendrelCathodeFrontAxisY.monitoring.maxVelocity := 2500.0;
   cmMendrelCathodeFrontAxisY.monitoring.actualCurrent := 0.0;
   cmMendrelCathodeFrontAxisY.monitoring.actualTorque := 0.0;
   cmMendrelCathodeFrontAxisY.monitoring.velocityOverrideEnabled := FALSE;
   cmMendrelCathodeFrontAxisY.monitoring.sinaParaError := FALSE;
   cmMendrelCathodeFrontAxisY.monitoring.sinaParaStatus := 16#0000_0000;
   cmMendrelCathodeFrontAxisY.configuration.referenceDesignator := WSTRING#'MendrelCathodeFrontAxisY';
   cmMendrelCathodeFrontAxisY.configuration.disableAlarms := FALSE;
   cmMendrelCathodeFrontAxisY.configuration.masterControlPopUp := TRUE;
   cmMendrelCathodeFrontAxisY.configuration.setPositions[0].position := 0.0;
   cmMendrelCathodeFrontAxisY.configuration.setPositions[1].position := 50.0;
   cmMendrelCathodeFrontAxisY.configuration.setPositions[2..15].position := 0.0;
   cmMendrelCathodeFrontAxisY.configuration.setPositions[0..1].velocity := 50.0;
   cmMendrelCathodeFrontAxisY.configuration.setPositions[2..15].velocity := -1.0;
   cmMendrelCathodeFrontAxisY.configuration.setPositions[0..1].acceleration := 500.0;
   cmMendrelCathodeFrontAxisY.configuration.setPositions[2..15].acceleration := -1.0;
   cmMendrelCathodeFrontAxisY.configuration.setPositions[0..1].deceleration := 500.0;
   cmMendrelCathodeFrontAxisY.configuration.setPositions[2..15].deceleration := -1.0;
   cmMendrelCathodeFrontAxisY.configuration.setPositions[0..15]."name" := '';
   cmMendrelCathodeFrontAxisZ.commandConfiguration.generalSettings.stopOnError := TRUE;
   cmMendrelCathodeFrontAxisZ.commandConfiguration.generalSettings.resetWithRestart := FALSE;
   cmMendrelCathodeFrontAxisZ.commandConfiguration.generalSettings.abortWaitingSyncCmd := TRUE;
   cmMendrelCathodeFrontAxisZ.commandConfiguration.power.startMode := 1;
   cmMendrelCathodeFrontAxisZ.commandConfiguration.power.stopMode := 0;
   cmMendrelCathodeFrontAxisZ.commandConfiguration.power.syncMotionSimulation := FALSE;
   cmMendrelCathodeFrontAxisZ.commandConfiguration.power.syncMotionSimulationExtendedMode := -1;
   cmMendrelCathodeFrontAxisZ.commandConfiguration.jog.velocity := 0.0;
   cmMendrelCathodeFrontAxisZ.commandConfiguration.jog.acceleration := -1.0;
   cmMendrelCathodeFrontAxisZ.commandConfiguration.jog.deceleration := -1.0;
   cmMendrelCathodeFrontAxisZ.commandConfiguration.jog.jerk := -1.0;
   cmMendrelCathodeFrontAxisZ.commandConfiguration.jog.positionControlled := TRUE;
   cmMendrelCathodeFrontAxisZ.commandConfiguration.jog.increment := 0.0;
   cmMendrelCathodeFrontAxisZ.commandConfiguration.jog.mode := 0;
   cmMendrelCathodeFrontAxisZ.commandConfiguration.moveVelocity.velocity := 0.0;
   cmMendrelCathodeFrontAxisZ.commandConfiguration.moveVelocity.acceleration := -1.0;
   cmMendrelCathodeFrontAxisZ.commandConfiguration.moveVelocity.deceleration := -1.0;
   cmMendrelCathodeFrontAxisZ.commandConfiguration.moveVelocity.jerk := -1.0;
   cmMendrelCathodeFrontAxisZ.commandConfiguration.moveVelocity.direction := 0;
   cmMendrelCathodeFrontAxisZ.commandConfiguration.moveVelocity.positionControlled := TRUE;
   cmMendrelCathodeFrontAxisZ.commandConfiguration.moveVelocity.velocityChangeOnTheFly := FALSE;
   cmMendrelCathodeFrontAxisZ.commandConfiguration.stop.deceleration := -1.0;
   cmMendrelCathodeFrontAxisZ.commandConfiguration.stop.jerk := -1.0;
   cmMendrelCathodeFrontAxisZ.commandConfiguration.stop.abortAcceleration := FALSE;
   cmMendrelCathodeFrontAxisZ.commandConfiguration.fastStop.deceleration := -1.0;
   cmMendrelCathodeFrontAxisZ.commandConfiguration.fastStop.jerk := -1.0;
   cmMendrelCathodeFrontAxisZ.commandConfiguration.fastStop.abortAcceleration := FALSE;
   cmMendrelCathodeFrontAxisZ.commandConfiguration.fastStop.replaceStopPossible := FALSE;
   cmMendrelCathodeFrontAxisZ.commandConfiguration.torqueLimiting.limit := -1.0;
   cmMendrelCathodeFrontAxisZ.commandConfiguration.torqueLimiting.mode := 0;
   cmMendrelCathodeFrontAxisZ.commandConfiguration.homing.position := 0.0;
   cmMendrelCathodeFrontAxisZ.commandConfiguration.homing.mode := 0;
   cmMendrelCathodeFrontAxisZ.commandConfiguration.homing.sensor := 0;
   cmMendrelCathodeFrontAxisZ.commandConfiguration.homing.extendedMode := -1;
   cmMendrelCathodeFrontAxisZ.commandConfiguration.homing.extendedModeTorqueLimit := 0.0;
   cmMendrelCathodeFrontAxisZ.commandConfiguration.homing.extendedModeTargetPosition := 0.0;
   cmMendrelCathodeFrontAxisZ.commandConfiguration.posRelative.distance := 0.0;
   cmMendrelCathodeFrontAxisZ.commandConfiguration.posRelative.velocity := -1.0;
   cmMendrelCathodeFrontAxisZ.commandConfiguration.posRelative.acceleration := -1.0;
   cmMendrelCathodeFrontAxisZ.commandConfiguration.posRelative.deceleration := -1.0;
   cmMendrelCathodeFrontAxisZ.commandConfiguration.posRelative.jerk := -1.0;
   cmMendrelCathodeFrontAxisZ.commandConfiguration.posRelative.direction := 0;
   cmMendrelCathodeFrontAxisZ.commandConfiguration.posAbsolute.position := 0.0;
   cmMendrelCathodeFrontAxisZ.commandConfiguration.posAbsolute.velocity := -1.0;
   cmMendrelCathodeFrontAxisZ.commandConfiguration.posAbsolute.acceleration := -1.0;
   cmMendrelCathodeFrontAxisZ.commandConfiguration.posAbsolute.deceleration := -1.0;
   cmMendrelCathodeFrontAxisZ.commandConfiguration.posAbsolute.jerk := -1.0;
   cmMendrelCathodeFrontAxisZ.commandConfiguration.posAbsolute.direction := 1;
   cmMendrelCathodeFrontAxisZ.commandConfiguration.posAbsolute.positionChangeOnTheFly := FALSE;
   cmMendrelCathodeFrontAxisZ.commandConfiguration.posAbsolute.velocityChangeOnTheFly := FALSE;
   cmMendrelCathodeFrontAxisZ.commandConfiguration.posSuperimposed.distance := 0.0;
   cmMendrelCathodeFrontAxisZ.commandConfiguration.posSuperimposed.velocityDiff := -1.0;
   cmMendrelCathodeFrontAxisZ.commandConfiguration.posSuperimposed.acceleration := -1.0;
   cmMendrelCathodeFrontAxisZ.commandConfiguration.posSuperimposed.deceleration := -1.0;
   cmMendrelCathodeFrontAxisZ.commandConfiguration.posSuperimposed.jerk := -1.0;
   cmMendrelCathodeFrontAxisZ.commandConfiguration.posSuperimposed.direction := 0;
   cmMendrelCathodeFrontAxisZ.commandConfiguration.haltSuperimposed.deceleration := -1.0;
   cmMendrelCathodeFrontAxisZ.commandConfiguration.haltSuperimposed.jerk := -1.0;
   cmMendrelCathodeFrontAxisZ.commandConfiguration.haltSuperimposed.abortAcceleration := FALSE;
   cmMendrelCathodeFrontAxisZ.commandConfiguration.gearInRelative.ratioNumerator := 1;
   cmMendrelCathodeFrontAxisZ.commandConfiguration.gearInRelative.ratioDenominator := 1;
   cmMendrelCathodeFrontAxisZ.commandConfiguration.gearInRelative.acceleration := -1.0;
   cmMendrelCathodeFrontAxisZ.commandConfiguration.gearInRelative.deceleration := -1.0;
   cmMendrelCathodeFrontAxisZ.commandConfiguration.gearInRelative.jerk := -1.0;
   cmMendrelCathodeFrontAxisZ.commandConfiguration.gearInRelative.ratioChangeOnTheFly := FALSE;
   cmMendrelCathodeFrontAxisZ.commandConfiguration.gearInAbsolute.ratioNumerator := 1;
   cmMendrelCathodeFrontAxisZ.commandConfiguration.gearInAbsolute.ratioDenominator := 1;
   cmMendrelCathodeFrontAxisZ.commandConfiguration.gearInAbsolute.masterSyncPosition := 0.0;
   cmMendrelCathodeFrontAxisZ.commandConfiguration.gearInAbsolute.slaveSyncPosition := 0.0;
   cmMendrelCathodeFrontAxisZ.commandConfiguration.gearInAbsolute.syncProfileReference := 1;
   cmMendrelCathodeFrontAxisZ.commandConfiguration.gearInAbsolute.masterStartDistance := 0.0;
   cmMendrelCathodeFrontAxisZ.commandConfiguration.gearInAbsolute.velocity := -1.0;
   cmMendrelCathodeFrontAxisZ.commandConfiguration.gearInAbsolute.acceleration := -1.0;
   cmMendrelCathodeFrontAxisZ.commandConfiguration.gearInAbsolute.deceleration := -1.0;
   cmMendrelCathodeFrontAxisZ.commandConfiguration.gearInAbsolute.jerk := -1.0;
   cmMendrelCathodeFrontAxisZ.commandConfiguration.gearInAbsolute.syncDirection := 1;
   cmMendrelCathodeFrontAxisZ.commandConfiguration.gearInAbsolute.ratioChangeOnTheFly := FALSE;
   cmMendrelCathodeFrontAxisZ.commandConfiguration.gearInVelocity.continuousUpdate := FALSE;
   cmMendrelCathodeFrontAxisZ.commandConfiguration.gearInVelocity.ratioNumerator := 1;
   cmMendrelCathodeFrontAxisZ.commandConfiguration.gearInVelocity.ratioDenominator := 1;
   cmMendrelCathodeFrontAxisZ.commandConfiguration.gearInVelocity.acceleration := -1.0;
   cmMendrelCathodeFrontAxisZ.commandConfiguration.gearInVelocity.deceleration := -1.0;
   cmMendrelCathodeFrontAxisZ.commandConfiguration.gearInVelocity.jerk := -1.0;
   cmMendrelCathodeFrontAxisZ.commandConfiguration.gearInVelocity.positionControlled := FALSE;
   cmMendrelCathodeFrontAxisZ.commandConfiguration.camIn.masterOffset := 0.0;
   cmMendrelCathodeFrontAxisZ.commandConfiguration.camIn.slaveOffset := 0.0;
   cmMendrelCathodeFrontAxisZ.commandConfiguration.camIn.masterScaling := 1.0;
   cmMendrelCathodeFrontAxisZ.commandConfiguration.camIn.slaveScaling := 1.0;
   cmMendrelCathodeFrontAxisZ.commandConfiguration.camIn.masterSyncPosition := 0.0;
   cmMendrelCathodeFrontAxisZ.commandConfiguration.camIn.syncProfileReference := 1;
   cmMendrelCathodeFrontAxisZ.commandConfiguration.camIn.masterStartDistance := 0.0;
   cmMendrelCathodeFrontAxisZ.commandConfiguration.camIn.velocity := -1.0;
   cmMendrelCathodeFrontAxisZ.commandConfiguration.camIn.acceleration := -1.0;
